SPLINE
SPL {X  -162.820, Y  +621.304, Z    +0.000, E1   +22.259, E3 +582034.378}
SPL {X  -162.820, Y  +618.758, Z    +0.000, E1   +22.239, E3 +582047.529}
SPL {X  -162.820, Y  +616.062, Z    +0.000, E1   +22.275, E3 +582060.950}
SPL {X  -162.820, Y  +613.536, Z    +0.000, E1   +22.242, E3 +582074.071}
SPL {X  -162.820, Y  +610.461, Z    +0.000, E1   +22.264, E3 +582089.703}
SPL {X  -162.820, Y  +606.755, Z    +0.000, E1   +22.275, E3 +582108.501}
SPL {X  -162.820, Y  +603.020, Z    +0.000, E1   +22.272, E3 +582127.561}
SPL {X  -162.820, Y  +599.168, Z    +0.000, E1   +22.310, E3 +582146.829}
SPL {X  -162.820, Y  +595.597, Z    +0.000, E1   +22.284, E3 +582165.165}
SPL {X  -162.820, Y  +593.320, Z    +0.000, E1   +22.199, E3 +582177.255}
SPL {X  -162.820, Y  +591.031, Z    +0.000, E1   +22.283, E3 +582188.346}
SPL {X  -162.820, Y  +588.026, Z    +0.000, E1   +22.301, E3 +582203.473}
SPL {X  -162.820, Y  +585.899, Z    +0.000, E1   +22.286, E3 +582214.275}
SPL {X  -162.820, Y  +583.204, Z    +0.000, E1   +22.278, E3 +582228.298}
SPL {X  -162.820, Y  +579.691, Z    +0.000, E1   +22.312, E3 +582245.786}
SPL {X  -162.820, Y  +576.856, Z    +0.000, E1   +22.233, E3 +582260.836}
SPL {X  -162.820, Y  +574.811, Z    +0.000, E1   +22.236, E3 +582271.100}
SPL {X  -162.820, Y  +572.645, Z    +0.000, E1   +22.246, E3 +582282.195}
SPL {X  -162.820, Y  +569.475, Z    +0.000, E1   +22.269, E3 +582298.202}
SPL {X  -162.820, Y  +565.838, Z    +0.000, E1   +22.271, E3 +582316.796}
SPL {X  -162.820, Y  +562.162, Z    +0.000, E1   +22.252, E3 +582335.614}
SPL {X  -162.820, Y  +558.919, Z    +0.000, E1   +22.286, E3 +582351.777}
SPL {X  -162.820, Y  +556.169, Z    +0.000, E1   +22.295, E3 +582365.606}
SPL {X  -162.820, Y  +553.294, Z    +0.000, E1   +22.266, E3 +582380.604}
SPL {X  -162.820, Y  +550.136, Z    +0.000, E1   +22.258, E3 +582396.717}
SPL {X  -162.820, Y  +546.694, Z    +0.000, E1   +22.290, E3 +582414.039}
SPL {X  -162.820, Y  +543.558, Z    +0.000, E1   +22.285, E3 +582429.902}
SPL {X  -162.820, Y  +541.633, Z    +0.000, E1   +22.257, E3 +582439.830}
SPL {X  -162.820, Y  +539.116, Z    +0.000, E1   +22.302, E3 +582452.441}
SPL {X  -162.820, Y  +535.523, Z    +0.000, E1   +22.266, E3 +582471.103}
SPL {X  -162.820, Y  +531.757, Z    +0.000, E1   +22.276, E3 +582490.157}
SPL {X  -162.820, Y  +527.980, Z    +0.000, E1   +22.326, E3 +582508.988}
SPL {X  -162.820, Y  +524.599, Z    +0.000, E1   +22.287, E3 +582526.385}
SPL {X  -162.820, Y  +522.011, Z    +0.000, E1   +22.282, E3 +582539.462}
SPL {X  -162.820, Y  +519.457, Z    +0.000, E1   +22.481, E3 +582550.752}
SPL {X  -162.820, Y  +505.859, Z    +0.000, E1   +28.367, E3 +582565.235}
SPL {X  -162.820, Y  +504.131, Z    +0.000, E1   +27.325, E3 +582579.373}
SPL {X  -162.820, Y  +503.215, Z    +0.000, E1   +26.369, E3 +582590.059}
SPL {X  -162.820, Y  +502.502, Z    +0.000, E1   +25.597, E3 +582598.906}
SPL {X  -162.820, Y  +501.672, Z    +0.000, E1   +24.583, E3 +582610.521}
SPL {X  -162.820, Y  +500.515, Z    +0.000, E1   +23.444, E3 +582625.051}
SPL {X  -162.820, Y  +499.633, Z    +0.000, E1   +22.486, E3 +582637.097}
SPL {X  -162.820, Y  +498.303, Z    +0.000, E1   +21.749, E3 +582650.406}
SPL {X  -162.820, Y  +495.897, Z    +0.000, E1   +21.662, E3 +582663.560}
SPL {X  -162.820, Y  +493.717, Z    +0.000, E1   +21.704, E3 +582674.666}
SPL {X  -162.820, Y  +491.396, Z    +0.000, E1   +21.707, E3 +582686.790}
SPL {X  -162.820, Y  +489.485, Z    +0.000, E1   +21.661, E3 +582697.138}
SPL {X  -162.820, Y  +487.723, Z    +0.000, E1   +21.665, E3 +582706.342}
SPL {X  -162.820, Y  +485.661, Z    +0.000, E1   +21.712, E3 +582716.785}
SPL {X  -162.820, Y  +482.775, Z    +0.000, E1   +21.716, E3 +582732.037}
SPL {X  -162.820, Y  +479.894, Z    +0.000, E1   +21.695, E3 +582747.114}
SPL {X  -162.820, Y  +477.685, Z    +0.000, E1   +21.656, E3 +582759.051}
SPL {X  -162.820, Y  +475.419, Z    +0.000, E1   +21.711, E3 +582770.404}
SPL {X  -162.820, Y  +473.301, Z    +0.000, E1   +21.712, E3 +582781.501}
SPL {X  -162.820, Y  +470.965, Z    +0.000, E1   +21.700, E3 +582793.846}
SPL {X  -162.820, Y  +469.036, Z    +0.000, E1   +21.695, E3 +582803.890}
SPL {X  -162.820, Y  +467.138, Z    +0.000, E1   +21.678, E3 +582814.061}
SPL {X  -162.820, Y  +465.011, Z    +0.000, E1   +21.692, E3 +582825.044}
SPL {X  -162.820, Y  +462.669, Z    +0.000, E1   +21.752, E3 +582836.824}
SPL {X  -162.820, Y  +460.725, Z    +0.000, E1   +21.689, E3 +582847.437}
SPL {X  -162.820, Y  +458.666, Z    +0.000, E1   +21.695, E3 +582858.249}
SPL {X  -162.820, Y  +456.431, Z    +0.000, E1   +21.708, E3 +582869.778}
SPL {X  -162.820, Y  +454.628, Z    +0.000, E1   +21.674, E3 +582879.496}
SPL {X  -162.820, Y  +452.690, Z    +0.000, E1   +21.773, E3 +582888.770}
SPL {X  -162.820, Y  +450.610, Z    +0.000, E1   +21.698, E3 +582900.369}
SPL {X  -162.820, Y  +448.170, Z    +0.000, E1   +21.667, E3 +582913.390}
SPL {X  -162.820, Y  +446.246, Z    +0.000, E1   +21.696, E3 +582923.208}
SPL {X  -162.820, Y  +443.784, Z    +0.000, E1   +21.713, E3 +582935.994}
SPL {X  -162.820, Y  +440.567, Z    +0.000, E1   +21.731, E3 +582952.834}
SPL {X  -162.820, Y  +437.628, Z    +0.000, E1   +21.678, E3 +582968.498}
SPL {X  -162.820, Y  +435.262, Z    +0.000, E1   +21.727, E3 +582980.433}
SPL {X  -162.820, Y  +433.510, Z    +0.000, E1   +21.692, E3 +582989.847}
SPL {X  -162.820, Y  +431.492, Z    +0.000, E1   +21.686, E3 +583000.543}
SPL {X  -162.820, Y  +429.074, Z    +0.000, E1   +21.710, E3 +583012.995}
SPL {X  -162.820, Y  +427.020, Z    +0.000, E1   +21.674, E3 +583023.996}
SPL {X  -162.820, Y  +424.525, Z    +0.000, E1   +21.712, E3 +583036.909}
SPL {X  -162.820, Y  +421.144, Z    +0.000, E1   +21.719, E3 +583054.576}
SPL {X  -162.820, Y  +418.116, Z    +0.000, E1   +21.761, E3 +583069.907}
SPL {X  -162.820, Y  +416.127, Z    +0.000, E1   +21.715, E3 +583080.612}
SPL {X  -162.820, Y  +414.361, Z    +0.000, E1   +21.613, E3 +583090.800}
SPL {X  -162.820, Y  +412.134, Z    +0.000, E1   +21.697, E3 +583101.744}
SPL {X  -162.820, Y  +409.248, Z    +0.000, E1   +21.741, E3 +583116.679}
SPL {X  -162.820, Y  +406.238, Z    +0.000, E1   +21.697, E3 +583132.647}
SPL {X  -162.820, Y  +404.001, Z    +0.000, E1   +21.723, E3 +583144.077}
SPL {X  -162.820, Y  +402.223, Z    +0.000, E1   +21.697, E3 +583153.562}
SPL {X  -162.820, Y  +400.348, Z    +0.000, E1   +21.713, E3 +583163.288}
SPL {X  -162.820, Y  +398.298, Z    +0.000, E1   +21.721, E3 +583173.904}
SPL {X  -162.820, Y  +396.371, Z    +0.000, E1   +21.713, E3 +583184.086}
SPL {X  -162.820, Y  +394.508, Z    +0.000, E1   +21.616, E3 +583194.641}
SPL {X  -162.820, Y  +392.435, Z    +0.000, E1   +21.681, E3 +583204.994}
SPL {X  -162.820, Y  +389.390, Z    +0.000, E1   +21.742, E3 +583220.601}
SPL {X  -162.820, Y  +386.818, Z    +0.000, E1   +21.679, E3 +583234.360}
SPL {X  -162.820, Y  +384.697, Z    +0.000, E1   +21.693, E3 +583245.430}
SPL {X  -162.820, Y  +382.288, Z    +0.000, E1   +21.742, E3 +583257.554}
SPL {X  -162.817, Y  +379.520, Z    +0.000, E1   +21.723, E3 +583272.391}
SPL {X  -162.776, Y  +376.710, Z    +0.000, E1   +21.698, E3 +583287.130}
SPL {X  -162.707, Y  +374.438, Z    +0.000, E1   +21.688, E3 +583299.134}
SPL {X  -162.607, Y  +372.171, Z    +0.000, E1   +21.692, E3 +583310.934}
SPL {X  -162.494, Y  +370.197, Z    +0.000, E1   +21.655, E3 +583321.560}
SPL {X  -162.349, Y  +368.131, Z    +0.000, E1   +21.624, E3 +583332.678}
SPL {X  -162.161, Y  +365.866, Z    +0.000, E1   +21.642, E3 +583344.363}
SPL {X  -161.651, Y  +361.024, Z    +0.000, E1   +22.970, E3 +583357.787}
SPL {X  -160.281, Y  +351.857, Z    +0.000, E1   +24.243, E3 +583393.126}
ENDSPLINE

SPLINE
SPL {X  -161.833, Y  +362.603, Z    +0.000, E1   +17.021, E3 +583407.822}
ENDSPLINE

SPLINE
SPL {X  -160.786, Y  +354.842, Z    +0.000, E1   +19.274, E3 +583439.977}
ENDSPLINE

SPLINE
SPL {X  -162.485, Y  +370.062, Z    +0.000, E1   +10.606, E3 +583446.355}
SPL {X  -162.818, Y  +379.636, Z    +0.000, E1    +5.115, E3 +583435.704}
SPL {X  -162.820, Y  +386.976, Z    +0.000, E1    +0.144, E3 +583434.803}
SPL {X  -162.820, Y  +391.982, Z    +0.000, E1    -3.443, E3 +583441.568}
SPL {X  -162.820, Y  +399.630, Z    +0.000, E1    -9.426, E3 +583444.076}
SPL {X  -162.820, Y  +408.127, Z    +0.000, E1   -18.417, E3 +583430.364}
SPL {X  -162.820, Y  +420.083, Z    +0.000, E1   -24.325, E3 +583450.839}
SPL {X  -162.820, Y  +428.527, Z    +0.000, E1   -26.988, E3 +583468.132}
SPL {X  -162.820, Y  +431.336, Z    +0.000, E1   -24.162, E3 +583498.342}
SPL {X  -162.820, Y  +432.048, Z    +0.000, E1   -22.832, E3 +583512.845}
SPL {X  -162.820, Y  +434.888, Z    +0.000, E1   -22.823, E3 +583526.795}
SPL {X  -162.820, Y  +436.834, Z    +0.000, E1   -22.779, E3 +583536.755}
SPL {X  -162.820, Y  +438.868, Z    +0.000, E1   -22.837, E3 +583546.408}
SPL {X  -162.820, Y  +441.351, Z    +0.000, E1   -22.805, E3 +583558.984}
SPL {X  -162.820, Y  +443.809, Z    +0.000, E1   -22.804, E3 +583571.150}
SPL {X  -162.820, Y  +446.105, Z    +0.000, E1   -22.815, E3 +583582.392}
SPL {X  -162.820, Y  +447.974, Z    +0.000, E1   -22.856, E3 +583591.295}
SPL {X  -162.820, Y  +449.911, Z    +0.000, E1   -22.774, E3 +583601.570}
SPL {X  -162.820, Y  +451.861, Z    +0.000, E1   -22.750, E3 +583611.417}
SPL {X  -162.820, Y  +454.167, Z    +0.000, E1   -22.842, E3 +583622.147}
SPL {X  -162.820, Y  +456.529, Z    +0.000, E1   -22.855, E3 +583633.675}
SPL {X  -162.820, Y  +458.725, Z    +0.000, E1   -22.793, E3 +583645.080}
SPL {X  -162.820, Y  +461.700, Z    +0.000, E1   -22.822, E3 +583659.702}
SPL {X  -162.820, Y  +464.633, Z    +0.000, E1   -22.813, E3 +583674.199}
SPL {X  -162.820, Y  +466.699, Z    +0.000, E1   -22.824, E3 +583684.245}
SPL {X  -162.820, Y  +468.655, Z    +0.000, E1   -22.858, E3 +583693.689}
SPL {X  -162.820, Y  +470.892, Z    +0.000, E1   -22.837, E3 +583704.927}
SPL {X  -162.820, Y  +473.485, Z    +0.000, E1   -22.806, E3 +583718.126}
SPL {X  -162.820, Y  +476.589, Z    +0.000, E1   -22.788, E3 +583733.648}
SPL {X  -162.820, Y  +478.914, Z    +0.000, E1   -22.821, E3 +583744.746}
SPL {X  -162.820, Y  +481.034, Z    +0.000, E1   -22.831, E3 +583755.268}
SPL {X  -162.820, Y  +484.256, Z    +0.000, E1   -22.840, E3 +583771.287}
SPL {X  -162.820, Y  +487.014, Z    +0.000, E1   -22.789, E3 +583785.154}
SPL {X  -162.820, Y  +489.750, Z    +0.000, E1   -22.832, E3 +583798.528}
SPL {X  -162.820, Y  +493.233, Z    +0.000, E1   -22.844, E3 +583815.665}
SPL {X  -162.820, Y  +496.150, Z    +0.000, E1   -22.796, E3 +583830.384}
SPL {X  -162.820, Y  +498.661, Z    +0.000, E1   -22.828, E3 +583842.565}
SPL {X  -162.820, Y  +501.761, Z    +0.000, E1   -22.820, E3 +583858.134}
SPL {X  -162.820, Y  +505.323, Z    +0.000, E1   -22.838, E3 +583875.581}
SPL {X  -162.820, Y  +507.875, Z    +0.000, E1   -22.849, E3 +583887.948}
SPL {X  -162.820, Y  +510.068, Z    +0.000, E1   -22.761, E3 +583899.641}
SPL {X  -162.820, Y  +512.359, Z    +0.000, E1   -22.823, E3 +583910.372}
SPL {X  -162.820, Y  +514.562, Z    +0.000, E1   -22.806, E3 +583921.559}
SPL {X  -162.820, Y  +517.952, Z    +0.000, E1   -22.864, E3 +583937.957}
SPL {X  -162.820, Y  +520.641, Z    +0.000, E1   -22.790, E3 +583951.675}
SPL {X  -162.820, Y  +522.740, Z    +0.000, E1   -22.811, E3 +583961.918}
SPL {X  -162.820, Y  +524.628, Z    +0.000, E1   -22.846, E3 +583970.913}
SPL {X  -162.820, Y  +526.661, Z    +0.000, E1   -22.801, E3 +583981.468}
SPL {X  -162.820, Y  +529.662, Z    +0.000, E1   -22.810, E3 +583996.319}
SPL {X  -162.820, Y  +532.614, Z    +0.000, E1   -22.828, E3 +584010.725}
SPL {X  -162.820, Y  +534.838, Z    +0.000, E1   -22.864, E3 +584021.354}
SPL {X  -162.820, Y  +536.882, Z    +0.000, E1   -22.782, E3 +584032.209}
SPL {X  -162.820, Y  +539.194, Z    +0.000, E1   -22.826, E3 +584043.257}
SPL {X  -162.820, Y  +541.555, Z    +0.000, E1   -22.817, E3 +584055.072}
SPL {X  -162.820, Y  +543.728, Z    +0.000, E1   -22.799, E3 +584065.929}
SPL {X  -162.820, Y  +545.925, Z    +0.000, E1   -22.803, E3 +584076.799}
SPL {X  -162.820, Y  +549.071, Z    +0.000, E1   -22.836, E3 +584092.326}
SPL {X  -162.820, Y  +553.089, Z    +0.000, E1   -22.838, E3 +584112.226}
SPL {X  -162.820, Y  +556.430, Z    +0.000, E1   -22.821, E3 +584128.728}
SPL {X  -162.820, Y  +558.974, Z    +0.000, E1   -22.806, E3 +584141.428}
SPL {X  -162.820, Y  +562.171, Z    +0.000, E1   -22.845, E3 +584157.126}
SPL {X  -162.820, Y  +565.170, Z    +0.000, E1   -22.801, E3 +584172.139}
SPL {X  -162.820, Y  +567.308, Z    +0.000, E1   -22.750, E3 +584183.155}
SPL {X  -162.820, Y  +570.378, Z    +0.000, E1   -22.843, E3 +584197.779}
SPL {X  -162.820, Y  +573.634, Z    +0.000, E1   -22.827, E3 +584213.923}
SPL {X  -162.820, Y  +576.228, Z    +0.000, E1   -22.814, E3 +584226.819}
SPL {X  -162.820, Y  +578.553, Z    +0.000, E1   -22.801, E3 +584238.435}
SPL {X  -162.820, Y  +581.064, Z    +0.000, E1   -22.823, E3 +584250.719}
SPL {X  -162.820, Y  +583.435, Z    +0.000, E1   -22.808, E3 +584262.541}
SPL {X  -162.820, Y  +585.410, Z    +0.000, E1   -22.764, E3 +584272.677}
SPL {X  -162.820, Y  +587.676, Z    +0.000, E1   -22.853, E3 +584283.191}
SPL {X  -162.820, Y  +590.707, Z    +0.000, E1   -22.855, E3 +584298.342}
SPL {X  -162.820, Y  +593.650, Z    +0.000, E1   -22.810, E3 +584313.102}
SPL {X  -162.820, Y  +595.830, Z    +0.000, E1   -22.828, E3 +584323.718}
SPL {X  -162.820, Y  +598.094, Z    +0.000, E1   -22.843, E3 +584334.831}
SPL {X  -162.820, Y  +600.420, Z    +0.000, E1   -22.826, E3 +584346.462}
SPL {X  -162.820, Y  +602.573, Z    +0.000, E1   -22.830, E3 +584357.047}
SPL {X  -162.820, Y  +604.828, Z    +0.000, E1   -22.784, E3 +584368.686}
SPL {X  -162.820, Y  +608.133, Z    +0.000, E1   -22.831, E3 +584384.803}
SPL {X  -162.820, Y  +611.103, Z    +0.000, E1   -22.785, E3 +584399.729}
SPL {X  -162.820, Y  +613.294, Z    +0.000, E1   -22.780, E3 +584410.602}
SPL {X  -162.820, Y  +615.356, Z    +0.000, E1   -22.799, E3 +584420.660}
SPL {X  -162.820, Y  +617.439, Z    +0.000, E1   -22.808, E3 +584430.918}
SPL {X  -162.820, Y  +619.665, Z    +0.000, E1   -22.817, E3 +584441.886}
SPL {X  -162.820, Y  +621.733, Z    +0.000, E1   -22.759, E3 +584452.610}
SPL {X  -162.820, Y  +624.076, Z    +0.000, E1   -22.774, E3 +584464.115}
SPL {X  -162.820, Y  +626.527, Z    +0.000, E1   -22.768, E3 +584476.358}
SPL {X  -162.820, Y  +629.758, Z    +0.000, E1   -22.800, E3 +584492.286}
SPL {X  -162.820, Y  +632.572, Z    +0.000, E1   -22.785, E3 +584506.136}
SPL {X  -162.820, Y  +634.507, Z    +0.000, E1   -22.784, E3 +584515.775}
SPL {X  -162.820, Y  +636.863, Z    +0.000, E1   -22.760, E3 +584527.697}
SPL {X  -162.820, Y  +639.254, Z    +0.000, E1   -22.767, E3 +584539.480}
SPL {X  -162.820, Y  +641.888, Z    +0.000, E1   -22.790, E3 +584552.427}
SPL {X  -162.820, Y  +644.915, Z    +0.000, E1   -22.818, E3 +584567.202}
SPL {X  -162.820, Y  +647.561, Z    +0.000, E1   -22.705, E3 +584581.244}
SPL {X  -162.820, Y  +649.758, Z    +0.000, E1   -22.780, E3 +584591.434}
SPL {X  -162.820, Y  +651.708, Z    +0.000, E1   -22.810, E3 +584600.929}
SPL {X  -162.820, Y  +653.898, Z    +0.000, E1   -22.796, E3 +584611.849}
SPL {X  -162.820, Y  +656.161, Z    +0.000, E1   -22.812, E3 +584622.971}
SPL {X  -162.820, Y  +658.384, Z    +0.000, E1   -22.822, E3 +584633.837}
SPL {X  -162.820, Y  +660.215, Z    +0.000, E1   -22.649, E3 +584644.428}
SPL {X  -162.820, Y  +662.823, Z    +0.000, E1   -22.799, E3 +584656.136}
SPL {X  -162.820, Y  +665.862, Z    +0.000, E1   -22.864, E3 +584670.835}
SPL {X  -162.820, Y  +668.960, Z    +0.000, E1   -22.773, E3 +584686.786}
SPL {X  -162.820, Y  +671.605, Z    +0.000, E1   -22.777, E3 +584699.860}
SPL {X  -162.817, Y  +674.515, Z    +0.000, E1   -22.816, E3 +584714.057}
SPL {X  -162.773, Y  +677.428, Z    +0.000, E1   -22.762, E3 +584728.865}
SPL {X  -162.691, Y  +679.987, Z    +0.000, E1   -22.794, E3 +584741.278}
SPL {X  -162.559, Y  +682.717, Z    +0.000, E1   -22.726, E3 +584755.461}
SPL {X  -162.404, Y  +685.137, Z    +0.000, E1   -22.766, E3 +584766.984}
SPL {X  -162.229, Y  +687.364, Z    +0.000, E1   -22.685, E3 +584778.852}
SPL {X  -161.938, Y  +690.422, Z    +0.000, E1   -22.769, E3 +584793.258}
SPL {X  -161.065, Y  +697.344, Z    +0.000, E1   -25.698, E3 +584802.378}
SPL {X  -158.553, Y  +710.529, Z    +0.000, E1   -30.890, E3 +584816.274}
ENDSPLINE

SPLINE
SPL {X  -161.215, Y  +696.305, Z    +0.000, E1   -20.575, E3 +584842.855}
SPL {X  -161.691, Y  +692.643, Z    +0.000, E1   -17.369, E3 +584859.043}
SPL {X  -162.534, Y  +683.153, Z    +0.000, E1   -10.475, E3 +584884.510}
SPL {X  -162.820, Y  +670.105, Z    +0.000, E1    -2.484, E3 +584877.157}
SPL {X  -162.820, Y  +665.819, Z    +0.000, E1    +0.492, E3 +584879.453}
SPL {X  -162.820, Y  +661.883, Z    +0.000, E1    +3.373, E3 +584883.930}
SPL {X  -162.820, Y  +655.163, Z    +0.000, E1    +8.702, E3 +584883.529}
SPL {X  -162.820, Y  +634.515, Z    +0.000, E1   +26.439, E3 +584875.942}
ENDSPLINE

SPLINE
SPL {X  -162.820, Y  +638.080, Z    +0.000, E1   +18.858, E3 +584905.906}
ENDSPLINE

SPLINE
SPL {X  -162.820, Y  +623.278, Z    +0.000, E1   +28.723, E3 +584907.477}
SPL {X  -162.820, Y  +611.829, Z    +0.000, E1   +31.229, E3 +584931.129}
ENDSPLINE

SPLINE
SPL {X  -162.820, Y  +623.595, Z    +0.000, E1   +22.712, E3 +584946.050}
ENDSPLINE

SPLINE
SPL {X  -162.820, Y  +621.304, Z    +0.000, E1   +22.259, E3 +584961.208}
SPL {X  -162.820, Y  +618.758, Z    +0.000, E1   +22.239, E3 +584974.358}
SPL {X  -162.820, Y  +616.062, Z    +0.000, E1   +22.275, E3 +584987.779}
SPL {X  -162.820, Y  +613.536, Z    +0.000, E1   +22.242, E3 +585000.901}
SPL {X  -162.820, Y  +611.128, Z    +0.000, E1   +22.252, E3 +585013.071}
SPL {X  -162.820, Y  +608.428, Z    +0.000, E1   +22.255, E3 +585026.855}
SPL {X  -162.820, Y  +605.178, Z    +0.000, E1   +22.267, E3 +585043.387}
SPL {X  -162.820, Y  +602.350, Z    +0.000, E1   +22.224, E3 +585058.004}
SPL {X  -162.820, Y  +599.842, Z    +0.000, E1   +22.298, E3 +585070.156}
SPL {X  -162.820, Y  +597.194, Z    +0.000, E1   +22.253, E3 +585084.077}
SPL {X  -162.820, Y  +594.779, Z    +0.000, E1   +22.284, E3 +585095.980}
SPL {X  -162.820, Y  +592.389, Z    +0.000, E1   +22.245, E3 +585108.597}
SPL {X  -162.820, Y  +589.492, Z    +0.000, E1   +22.304, E3 +585122.781}
SPL {X  -162.820, Y  +587.447, Z    +0.000, E1   +22.279, E3 +585133.310}
SPL {X  -162.820, Y  +585.192, Z    +0.000, E1   +22.298, E3 +585144.721}
SPL {X  -162.820, Y  +582.610, Z    +0.000, E1   +22.234, E3 +585158.344}
SPL {X  -162.820, Y  +580.317, Z    +0.000, E1   +22.300, E3 +585169.398}
SPL {X  -162.820, Y  +578.878, Z    +0.000, E1   +22.272, E3 +585176.907}
SPL {X  -162.820, Y  +576.856, Z    +0.000, E1   +22.233, E3 +585187.666}
SPL {X  -162.820, Y  +574.811, Z    +0.000, E1   +22.236, E3 +585197.929}
SPL {X  -162.820, Y  +572.645, Z    +0.000, E1   +22.246, E3 +585209.025}
SPL {X  -162.820, Y  +569.475, Z    +0.000, E1   +22.269, E3 +585225.031}
SPL {X  -162.820, Y  +565.838, Z    +0.000, E1   +22.271, E3 +585243.626}
SPL {X  -162.820, Y  +562.162, Z    +0.000, E1   +22.252, E3 +585262.443}
SPL {X  -162.820, Y  +558.919, Z    +0.000, E1   +22.286, E3 +585278.606}
SPL {X  -162.820, Y  +556.169, Z    +0.000, E1   +22.295, E3 +585292.436}
SPL {X  -162.820, Y  +553.294, Z    +0.000, E1   +22.266, E3 +585307.433}
SPL {X  -162.820, Y  +550.136, Z    +0.000, E1   +22.258, E3 +585323.546}
SPL {X  -162.820, Y  +546.694, Z    +0.000, E1   +22.290, E3 +585340.868}
SPL {X  -162.820, Y  +543.558, Z    +0.000, E1   +22.285, E3 +585356.731}
SPL {X  -162.820, Y  +541.633, Z    +0.000, E1   +22.257, E3 +585366.659}
SPL {X  -162.820, Y  +539.116, Z    +0.000, E1   +22.302, E3 +585379.270}
SPL {X  -162.820, Y  +536.913, Z    +0.000, E1   +22.192, E3 +585391.195}
SPL {X  -162.820, Y  +534.880, Z    +0.000, E1   +22.252, E3 +585401.148}
SPL {X  -162.820, Y  +532.896, Z    +0.000, E1   +22.234, E3 +585411.308}
SPL {X  -162.820, Y  +531.056, Z    +0.000, E1   +22.251, E3 +585420.590}
SPL {X  -162.820, Y  +528.708, Z    +0.000, E1   +22.319, E3 +585431.972}
SPL {X  -162.820, Y  +525.932, Z    +0.000, E1   +22.258, E3 +585446.728}
SPL {X  -162.820, Y  +522.524, Z    +0.000, E1   +22.326, E3 +585463.452}
SPL {X  -162.820, Y  +519.457, Z    +0.000, E1   +22.481, E3 +585477.581}
SPL {X  -162.820, Y  +506.285, Z    +0.000, E1   +28.538, E3 +585489.039}
SPL {X  -162.820, Y  +504.441, Z    +0.000, E1   +27.574, E3 +585503.381}
SPL {X  -162.820, Y  +502.813, Z    +0.000, E1   +26.013, E3 +585521.579}
SPL {X  -162.820, Y  +502.016, Z    +0.000, E1   +24.802, E3 +585533.921}
SPL {X  -162.820, Y  +501.060, Z    +0.000, E1   +24.081, E3 +585544.111}
SPL {X  -162.820, Y  +500.336, Z    +0.000, E1   +23.110, E3 +585555.251}
SPL {X  -162.820, Y  +499.240, Z    +0.000, E1   +22.316, E3 +585567.561}
SPL {X  -162.820, Y  +498.027, Z    +0.000, E1   +21.516, E3 +585580.469}
SPL {X  -162.820, Y  +495.897, Z    +0.000, E1   +21.662, E3 +585590.389}
SPL {X  -162.820, Y  +493.717, Z    +0.000, E1   +21.704, E3 +585601.496}
SPL {X  -162.820, Y  +491.396, Z    +0.000, E1   +21.707, E3 +585613.620}
SPL {X  -162.820, Y  +488.560, Z    +0.000, E1   +21.695, E3 +585628.729}
SPL {X  -162.820, Y  +485.661, Z    +0.000, E1   +21.712, E3 +585643.614}
SPL {X  -162.820, Y  +483.668, Z    +0.000, E1   +21.664, E3 +585654.442}
SPL {X  -162.820, Y  +481.739, Z    +0.000, E1   +21.704, E3 +585664.156}
SPL {X  -162.820, Y  +479.894, Z    +0.000, E1   +21.695, E3 +585673.943}
SPL {X  -162.820, Y  +477.685, Z    +0.000, E1   +21.656, E3 +585685.881}
SPL {X  -162.820, Y  +475.419, Z    +0.000, E1   +21.711, E3 +585697.233}
SPL {X  -162.820, Y  +473.301, Z    +0.000, E1   +21.712, E3 +585708.330}
SPL {X  -162.820, Y  +470.965, Z    +0.000, E1   +21.700, E3 +585720.675}
SPL {X  -162.820, Y  +469.036, Z    +0.000, E1   +21.695, E3 +585730.719}
SPL {X  -162.820, Y  +467.138, Z    +0.000, E1   +21.678, E3 +585740.891}
SPL {X  -162.820, Y  +465.011, Z    +0.000, E1   +21.692, E3 +585751.873}
SPL {X  -162.820, Y  +462.669, Z    +0.000, E1   +21.752, E3 +585763.654}
SPL {X  -162.820, Y  +460.725, Z    +0.000, E1   +21.689, E3 +585774.267}
SPL {X  -162.820, Y  +458.666, Z    +0.000, E1   +21.695, E3 +585785.079}
SPL {X  -162.820, Y  +456.431, Z    +0.000, E1   +21.708, E3 +585796.607}
SPL {X  -162.820, Y  +453.609, Z    +0.000, E1   +21.757, E3 +585811.141}
SPL {X  -162.820, Y  +450.610, Z    +0.000, E1   +21.698, E3 +585827.198}
SPL {X  -162.820, Y  +448.170, Z    +0.000, E1   +21.667, E3 +585840.219}
SPL {X  -162.820, Y  +446.246, Z    +0.000, E1   +21.696, E3 +585850.037}
SPL {X  -162.820, Y  +443.784, Z    +0.000, E1   +21.713, E3 +585862.823}
SPL {X  -162.820, Y  +440.567, Z    +0.000, E1   +21.731, E3 +585879.663}
SPL {X  -162.820, Y  +437.628, Z    +0.000, E1   +21.678, E3 +585895.327}
SPL {X  -162.820, Y  +434.473, Z    +0.000, E1   +21.747, E3 +585911.423}
SPL {X  -162.820, Y  +431.492, Z    +0.000, E1   +21.686, E3 +585927.372}
SPL {X  -162.820, Y  +429.074, Z    +0.000, E1   +21.710, E3 +585939.824}
SPL {X  -162.820, Y  +426.023, Z    +0.000, E1   +21.718, E3 +585955.892}
SPL {X  -162.820, Y  +422.986, Z    +0.000, E1   +21.685, E3 +585971.939}
SPL {X  -162.820, Y  +420.528, Z    +0.000, E1   +21.706, E3 +585984.589}
SPL {X  -162.820, Y  +418.116, Z    +0.000, E1   +21.761, E3 +585996.736}
SPL {X  -162.820, Y  +416.127, Z    +0.000, E1   +21.715, E3 +586007.442}
SPL {X  -162.820, Y  +414.361, Z    +0.000, E1   +21.613, E3 +586017.629}
SPL {X  -162.820, Y  +411.450, Z    +0.000, E1   +21.710, E3 +586032.202}
SPL {X  -162.820, Y  +408.590, Z    +0.000, E1   +21.735, E3 +586046.828}
SPL {X  -162.820, Y  +406.238, Z    +0.000, E1   +21.697, E3 +586059.477}
SPL {X  -162.820, Y  +403.166, Z    +0.000, E1   +21.746, E3 +586075.283}
SPL {X  -162.820, Y  +400.348, Z    +0.000, E1   +21.713, E3 +586090.117}
SPL {X  -162.820, Y  +398.298, Z    +0.000, E1   +21.721, E3 +586100.733}
SPL {X  -162.820, Y  +396.371, Z    +0.000, E1   +21.713, E3 +586110.915}
SPL {X  -162.820, Y  +394.508, Z    +0.000, E1   +21.616, E3 +586121.470}
SPL {X  -162.820, Y  +391.777, Z    +0.000, E1   +21.714, E3 +586135.130}
SPL {X  -162.820, Y  +388.822, Z    +0.000, E1   +21.717, E3 +586150.449}
SPL {X  -162.820, Y  +386.818, Z    +0.000, E1   +21.679, E3 +586161.189}
SPL {X  -162.820, Y  +384.697, Z    +0.000, E1   +21.693, E3 +586172.260}
SPL {X  -162.820, Y  +382.288, Z    +0.000, E1   +21.742, E3 +586184.383}
SPL {X  -162.820, Y  +380.381, Z    +0.000, E1   +21.655, E3 +586195.108}
SPL {X  -162.808, Y  +378.512, Z    +0.000, E1   +21.736, E3 +586204.160}
SPL {X  -162.776, Y  +376.710, Z    +0.000, E1   +21.698, E3 +586213.960}
SPL {X  -162.707, Y  +374.438, Z    +0.000, E1   +21.688, E3 +586225.964}
SPL {X  -162.607, Y  +372.171, Z    +0.000, E1   +21.692, E3 +586237.763}
SPL {X  -162.494, Y  +370.197, Z    +0.000, E1   +21.655, E3 +586248.389}
SPL {X  -162.349, Y  +368.131, Z    +0.000, E1   +21.624, E3 +586259.507}
SPL {X  -162.161, Y  +365.866, Z    +0.000, E1   +21.642, E3 +586271.193}
SPL {X  -161.651, Y  +361.024, Z    +0.000, E1   +22.970, E3 +586284.616}
SPL {X  -160.281, Y  +351.857, Z    +0.000, E1   +24.243, E3 +586319.955}
ENDSPLINE

SPLINE
SPL {X  -161.833, Y  +362.603, Z    +0.000, E1   +17.021, E3 +586334.651}
ENDSPLINE

SPLINE
SPL {X  -160.786, Y  +354.842, Z    +0.000, E1   +19.274, E3 +586366.806}
ENDSPLINE

SPLINE
SPL {X  -162.485, Y  +370.062, Z    +0.000, E1   +10.606, E3 +586373.185}
SPL {X  -162.818, Y  +379.636, Z    +0.000, E1    +5.115, E3 +586362.534}
SPL {X  -162.820, Y  +386.976, Z    +0.000, E1    +0.144, E3 +586361.633}
SPL {X  -162.820, Y  +391.982, Z    +0.000, E1    -3.443, E3 +586368.397}
SPL {X  -162.820, Y  +399.630, Z    +0.000, E1    -9.426, E3 +586370.905}
SPL {X  -162.820, Y  +408.127, Z    +0.000, E1   -18.417, E3 +586357.193}
SPL {X  -162.820, Y  +420.083, Z    +0.000, E1   -24.325, E3 +586377.669}
SPL {X  -162.820, Y  +428.527, Z    +0.000, E1   -26.988, E3 +586394.961}
SPL {X  -162.820, Y  +431.191, Z    +0.000, E1   -23.548, E3 +586429.814}
SPL {X  -162.820, Y  +432.946, Z    +0.000, E1   -22.795, E3 +586444.217}
SPL {X  -162.820, Y  +434.888, Z    +0.000, E1   -22.823, E3 +586453.624}
SPL {X  -162.820, Y  +436.834, Z    +0.000, E1   -22.779, E3 +586463.584}
SPL {X  -162.820, Y  +438.868, Z    +0.000, E1   -22.837, E3 +586473.238}
SPL {X  -162.820, Y  +441.351, Z    +0.000, E1   -22.805, E3 +586485.813}
SPL {X  -162.820, Y  +443.809, Z    +0.000, E1   -22.804, E3 +586497.979}
SPL {X  -162.820, Y  +447.077, Z    +0.000, E1   -22.869, E3 +586513.790}
SPL {X  -162.820, Y  +449.911, Z    +0.000, E1   -22.774, E3 +586528.399}
SPL {X  -162.820, Y  +451.861, Z    +0.000, E1   -22.750, E3 +586538.247}
SPL {X  -162.820, Y  +454.167, Z    +0.000, E1   -22.842, E3 +586548.976}
SPL {X  -162.820, Y  +456.529, Z    +0.000, E1   -22.855, E3 +586560.505}
SPL {X  -162.820, Y  +458.725, Z    +0.000, E1   -22.793, E3 +586571.909}
SPL {X  -162.820, Y  +461.700, Z    +0.000, E1   -22.822, E3 +586586.532}
SPL {X  -162.820, Y  +464.633, Z    +0.000, E1   -22.813, E3 +586601.028}
SPL {X  -162.820, Y  +466.699, Z    +0.000, E1   -22.824, E3 +586611.074}
SPL {X  -162.820, Y  +468.655, Z    +0.000, E1   -22.858, E3 +586620.518}
SPL {X  -162.820, Y  +470.892, Z    +0.000, E1   -22.837, E3 +586631.757}
SPL {X  -162.820, Y  +473.485, Z    +0.000, E1   -22.806, E3 +586644.955}
SPL {X  -162.820, Y  +475.738, Z    +0.000, E1   -22.728, E3 +586656.620}
SPL {X  -162.820, Y  +478.177, Z    +0.000, E1   -22.834, E3 +586667.960}
SPL {X  -162.820, Y  +481.034, Z    +0.000, E1   -22.831, E3 +586682.097}
SPL {X  -162.820, Y  +483.391, Z    +0.000, E1   -22.793, E3 +586694.033}
SPL {X  -162.820, Y  +486.307, Z    +0.000, E1   -22.833, E3 +586708.287}
SPL {X  -162.820, Y  +489.750, Z    +0.000, E1   -22.832, E3 +586725.357}
SPL {X  -162.820, Y  +492.546, Z    +0.000, E1   -22.823, E3 +586739.115}
SPL {X  -162.820, Y  +495.526, Z    +0.000, E1   -22.833, E3 +586753.998}
SPL {X  -162.820, Y  +499.330, Z    +0.000, E1   -22.841, E3 +586772.779}
SPL {X  -162.820, Y  +503.049, Z    +0.000, E1   -22.823, E3 +586791.329}
SPL {X  -162.820, Y  +506.908, Z    +0.000, E1   -22.877, E3 +586809.999}
SPL {X  -162.820, Y  +510.068, Z    +0.000, E1   -22.761, E3 +586826.470}
SPL {X  -162.820, Y  +512.359, Z    +0.000, E1   -22.823, E3 +586837.202}
SPL {X  -162.820, Y  +513.873, Z    +0.000, E1   -22.800, E3 +586844.888}
SPL {X  -162.820, Y  +516.100, Z    +0.000, E1   -22.809, E3 +586855.965}
SPL {X  -162.820, Y  +518.662, Z    +0.000, E1   -22.847, E3 +586868.263}
SPL {X  -162.820, Y  +520.641, Z    +0.000, E1   -22.790, E3 +586878.504}
SPL {X  -162.820, Y  +523.535, Z    +0.000, E1   -22.857, E3 +586892.473}
SPL {X  -162.820, Y  +526.661, Z    +0.000, E1   -22.801, E3 +586908.297}
SPL {X  -162.820, Y  +528.725, Z    +0.000, E1   -22.770, E3 +586918.667}
SPL {X  -162.820, Y  +530.303, Z    +0.000, E1   -22.798, E3 +586926.286}
SPL {X  -162.820, Y  +532.614, Z    +0.000, E1   -22.828, E3 +586937.554}
SPL {X  -162.820, Y  +534.838, Z    +0.000, E1   -22.864, E3 +586948.183}
SPL {X  -162.820, Y  +536.882, Z    +0.000, E1   -22.782, E3 +586959.038}
SPL {X  -162.820, Y  +539.194, Z    +0.000, E1   -22.826, E3 +586970.087}
SPL {X  -162.820, Y  +541.555, Z    +0.000, E1   -22.817, E3 +586981.901}
SPL {X  -162.820, Y  +543.728, Z    +0.000, E1   -22.799, E3 +586992.758}
SPL {X  -162.820, Y  +545.925, Z    +0.000, E1   -22.803, E3 +587003.628}
SPL {X  -162.820, Y  +548.328, Z    +0.000, E1   -22.796, E3 +587015.624}
SPL {X  -162.820, Y  +551.027, Z    +0.000, E1   -22.819, E3 +587028.817}
SPL {X  -162.820, Y  +553.721, Z    +0.000, E1   -22.807, E3 +587042.261}
SPL {X  -162.820, Y  +556.430, Z    +0.000, E1   -22.821, E3 +587055.557}
SPL {X  -162.820, Y  +559.675, Z    +0.000, E1   -22.837, E3 +587071.637}
SPL {X  -162.820, Y  +562.799, Z    +0.000, E1   -22.814, E3 +587087.143}
SPL {X  -162.820, Y  +565.170, Z    +0.000, E1   -22.801, E3 +587098.968}
SPL {X  -162.820, Y  +568.020, Z    +0.000, E1   -22.787, E3 +587113.355}
SPL {X  -162.820, Y  +570.992, Z    +0.000, E1   -22.834, E3 +587127.574}
SPL {X  -162.820, Y  +572.901, Z    +0.000, E1   -22.775, E3 +587137.442}
SPL {X  -162.820, Y  +575.638, Z    +0.000, E1   -22.855, E3 +587150.552}
SPL {X  -162.820, Y  +578.553, Z    +0.000, E1   -22.801, E3 +587165.264}
SPL {X  -162.820, Y  +581.064, Z    +0.000, E1   -22.823, E3 +587177.549}
SPL {X  -162.820, Y  +583.435, Z    +0.000, E1   -22.808, E3 +587189.370}
SPL {X  -162.820, Y  +585.410, Z    +0.000, E1   -22.764, E3 +587199.506}
SPL {X  -162.820, Y  +587.676, Z    +0.000, E1   -22.853, E3 +587210.021}
SPL {X  -162.820, Y  +589.682, Z    +0.000, E1   -22.776, E3 +587220.551}
SPL {X  -162.820, Y  +591.720, Z    +0.000, E1   -22.868, E3 +587229.861}
SPL {X  -162.820, Y  +593.650, Z    +0.000, E1   -22.810, E3 +587239.931}
SPL {X  -162.820, Y  +595.830, Z    +0.000, E1   -22.828, E3 +587250.547}
SPL {X  -162.820, Y  +598.094, Z    +0.000, E1   -22.843, E3 +587261.660}
SPL {X  -162.820, Y  +600.420, Z    +0.000, E1   -22.826, E3 +587273.291}
SPL {X  -162.820, Y  +602.573, Z    +0.000, E1   -22.830, E3 +587283.877}
SPL {X  -162.820, Y  +604.828, Z    +0.000, E1   -22.784, E3 +587295.515}
SPL {X  -162.820, Y  +608.133, Z    +0.000, E1   -22.831, E3 +587311.633}
SPL {X  -162.820, Y  +611.103, Z    +0.000, E1   -22.785, E3 +587326.558}
SPL {X  -162.820, Y  +613.294, Z    +0.000, E1   -22.780, E3 +587337.432}
SPL {X  -162.820, Y  +615.356, Z    +0.000, E1   -22.799, E3 +587347.489}
SPL {X  -162.820, Y  +617.439, Z    +0.000, E1   -22.808, E3 +587357.747}
SPL {X  -162.820, Y  +619.665, Z    +0.000, E1   -22.817, E3 +587368.715}
SPL {X  -162.820, Y  +621.733, Z    +0.000, E1   -22.759, E3 +587379.439}
SPL {X  -162.820, Y  +624.076, Z    +0.000, E1   -22.774, E3 +587390.944}
SPL {X  -162.820, Y  +627.244, Z    +0.000, E1   -22.803, E3 +587406.627}
SPL {X  -162.820, Y  +630.349, Z    +0.000, E1   -22.766, E3 +587422.158}
SPL {X  -162.820, Y  +632.572, Z    +0.000, E1   -22.785, E3 +587432.965}
SPL {X  -162.820, Y  +634.507, Z    +0.000, E1   -22.784, E3 +587442.604}
SPL {X  -162.820, Y  +636.863, Z    +0.000, E1   -22.760, E3 +587454.526}
SPL {X  -162.820, Y  +639.254, Z    +0.000, E1   -22.767, E3 +587466.309}
SPL {X  -162.820, Y  +641.195, Z    +0.000, E1   -22.782, E3 +587475.757}
SPL {X  -162.820, Y  +643.449, Z    +0.000, E1   -22.796, E3 +587486.927}
SPL {X  -162.820, Y  +645.630, Z    +0.000, E1   -22.795, E3 +587497.623}
SPL {X  -162.820, Y  +647.561, Z    +0.000, E1   -22.705, E3 +587508.073}
SPL {X  -162.820, Y  +651.051, Z    +0.000, E1   -22.833, E3 +587524.493}
SPL {X  -162.820, Y  +653.898, Z    +0.000, E1   -22.796, E3 +587538.679}
SPL {X  -162.820, Y  +656.161, Z    +0.000, E1   -22.812, E3 +587549.800}
SPL {X  -162.820, Y  +658.384, Z    +0.000, E1   -22.822, E3 +587560.666}
SPL {X  -162.820, Y  +660.215, Z    +0.000, E1   -22.649, E3 +587571.257}
SPL {X  -162.820, Y  +662.823, Z    +0.000, E1   -22.799, E3 +587582.965}
SPL {X  -162.820, Y  +665.112, Z    +0.000, E1   -22.835, E3 +587594.019}
SPL {X  -162.820, Y  +667.016, Z    +0.000, E1   -22.823, E3 +587603.448}
SPL {X  -162.820, Y  +668.960, Z    +0.000, E1   -22.773, E3 +587613.615}
SPL {X  -162.820, Y  +671.605, Z    +0.000, E1   -22.777, E3 +587626.689}
SPL {X  -162.817, Y  +674.515, Z    +0.000, E1   -22.816, E3 +587640.886}
SPL {X  -162.773, Y  +677.428, Z    +0.000, E1   -22.762, E3 +587655.694}
SPL {X  -162.691, Y  +679.987, Z    +0.000, E1   -22.794, E3 +587668.107}
SPL {X  -162.604, Y  +681.880, Z    +0.000, E1   -22.691, E3 +587678.268}
SPL {X  -162.458, Y  +684.346, Z    +0.000, E1   -22.764, E3 +587690.062}
SPL {X  -162.296, Y  +686.547, Z    +0.000, E1   -22.660, E3 +587701.678}
SPL {X  -162.090, Y  +688.902, Z    +0.000, E1   -22.700, E3 +587713.187}
SPL {X  -161.474, Y  +694.390, Z    +0.000, E1   -24.298, E3 +587726.542}
SPL {X  -158.730, Y  +709.763, Z    +0.000, E1   -31.225, E3 +587737.880}
ENDSPLINE

SPLINE
SPL {X  -160.932, Y  +698.225, Z    +0.000, E1   -21.712, E3 +587768.990}
SPL {X  -161.691, Y  +692.643, Z    +0.000, E1   -17.369, E3 +587785.873}
SPL {X  -162.534, Y  +683.153, Z    +0.000, E1   -10.475, E3 +587811.340}
SPL {X  -162.820, Y  +670.105, Z    +0.000, E1    -2.484, E3 +587803.986}
SPL {X  -162.820, Y  +665.819, Z    +0.000, E1    +0.492, E3 +587806.283}
SPL {X  -162.820, Y  +661.883, Z    +0.000, E1    +3.373, E3 +587810.759}
SPL {X  -162.820, Y  +653.808, Z    +0.000, E1    +9.891, E3 +587808.450}
SPL {X  -162.820, Y  +632.548, Z    +0.000, E1   +27.446, E3 +587804.987}
ENDSPLINE

SPLINE
SPL {X  -162.820, Y  +638.080, Z    +0.000, E1   +18.858, E3 +587832.736}
ENDSPLINE

SPLINE
SPL {X  -162.820, Y  +623.278, Z    +0.000, E1   +28.723, E3 +587834.306}
SPL {X  -162.820, Y  +611.829, Z    +0.000, E1   +31.229, E3 +587857.958}
ENDSPLINE

SPLINE
SPL {X  -162.820, Y  +623.595, Z    +0.000, E1   +22.712, E3 +587872.879}
ENDSPLINE

SPLINE
SPL {X  -162.820, Y  +621.304, Z    +0.000, E1   +22.259, E3 +587888.037}
SPL {X  -162.820, Y  +618.758, Z    +0.000, E1   +22.239, E3 +587901.188}
SPL {X  -162.820, Y  +616.062, Z    +0.000, E1   +22.275, E3 +587914.608}
SPL {X  -162.820, Y  +613.536, Z    +0.000, E1   +22.242, E3 +587927.730}
SPL {X  -162.820, Y  +610.461, Z    +0.000, E1   +22.264, E3 +587943.361}
SPL {X  -162.820, Y  +606.755, Z    +0.000, E1   +22.275, E3 +587962.159}
SPL {X  -162.820, Y  +603.020, Z    +0.000, E1   +22.272, E3 +587981.219}
SPL {X  -162.820, Y  +599.168, Z    +0.000, E1   +22.310, E3 +588000.487}
SPL {X  -162.820, Y  +596.569, Z    +0.000, E1   +22.222, E3 +588014.209}
SPL {X  -162.820, Y  +594.115, Z    +0.000, E1   +22.273, E3 +588026.435}
SPL {X  -162.820, Y  +591.721, Z    +0.000, E1   +22.239, E3 +588038.750}
SPL {X  -162.820, Y  +589.492, Z    +0.000, E1   +22.304, E3 +588049.611}
SPL {X  -162.820, Y  +586.660, Z    +0.000, E1   +22.307, E3 +588064.051}
SPL {X  -162.820, Y  +583.204, Z    +0.000, E1   +22.278, E3 +588081.956}
SPL {X  -162.820, Y  +580.317, Z    +0.000, E1   +22.300, E3 +588096.227}
SPL {X  -162.820, Y  +578.061, Z    +0.000, E1   +22.264, E3 +588108.112}
SPL {X  -162.820, Y  +575.394, Z    +0.000, E1   +22.240, E3 +588121.857}
SPL {X  -162.820, Y  +573.156, Z    +0.000, E1   +22.254, E3 +588133.066}
SPL {X  -162.820, Y  +570.852, Z    +0.000, E1   +22.234, E3 +588145.090}
SPL {X  -162.820, Y  +567.961, Z    +0.000, E1   +22.247, E3 +588159.694}
SPL {X  -162.820, Y  +564.506, Z    +0.000, E1   +22.298, E3 +588177.008}
SPL {X  -162.820, Y  +561.620, Z    +0.000, E1   +22.191, E3 +588192.389}
SPL {X  -162.820, Y  +559.515, Z    +0.000, E1   +22.273, E3 +588202.391}
SPL {X  -162.820, Y  +556.723, Z    +0.000, E1   +22.309, E3 +588216.475}
SPL {X  -162.820, Y  +553.294, Z    +0.000, E1   +22.266, E3 +588234.262}
SPL {X  -162.820, Y  +550.871, Z    +0.000, E1   +22.229, E3 +588246.736}
SPL {X  -162.820, Y  +548.168, Z    +0.000, E1   +22.298, E3 +588260.073}
SPL {X  -162.820, Y  +545.860, Z    +0.000, E1   +22.216, E3 +588272.330}
SPL {X  -162.820, Y  +543.558, Z    +0.000, E1   +22.285, E3 +588283.561}
SPL {X  -162.820, Y  +540.968, Z    +0.000, E1   +22.274, E3 +588296.833}
SPL {X  -162.820, Y  +538.512, Z    +0.000, E1   +22.287, E3 +588309.145}
SPL {X  -162.820, Y  +535.523, Z    +0.000, E1   +22.266, E3 +588324.761}
SPL {X  -162.820, Y  +531.757, Z    +0.000, E1   +22.276, E3 +588343.816}
SPL {X  -162.820, Y  +527.980, Z    +0.000, E1   +22.326, E3 +588362.647}
SPL {X  -162.820, Y  +524.599, Z    +0.000, E1   +22.287, E3 +588380.044}
SPL {X  -162.820, Y  +522.011, Z    +0.000, E1   +22.282, E3 +588393.121}
SPL {X  -162.820, Y  +519.457, Z    +0.000, E1   +22.481, E3 +588404.410}
SPL {X  -162.820, Y  +505.859, Z    +0.000, E1   +28.367, E3 +588418.893}
SPL {X  -162.820, Y  +504.131, Z    +0.000, E1   +27.325, E3 +588433.032}
SPL {X  -162.820, Y  +503.215, Z    +0.000, E1   +26.369, E3 +588443.718}
SPL {X  -162.820, Y  +502.265, Z    +0.000, E1   +25.287, E3 +588456.200}
SPL {X  -162.820, Y  +501.060, Z    +0.000, E1   +24.081, E3 +588470.940}
SPL {X  -162.820, Y  +500.336, Z    +0.000, E1   +23.110, E3 +588482.080}
SPL {X  -162.820, Y  +499.240, Z    +0.000, E1   +22.316, E3 +588494.391}
SPL {X  -162.820, Y  +498.027, Z    +0.000, E1   +21.516, E3 +588507.298}
SPL {X  -162.820, Y  +495.897, Z    +0.000, E1   +21.662, E3 +588517.219}
SPL {X  -162.820, Y  +493.717, Z    +0.000, E1   +21.704, E3 +588528.325}
SPL {X  -162.820, Y  +491.396, Z    +0.000, E1   +21.707, E3 +588540.449}
SPL {X  -162.820, Y  +488.560, Z    +0.000, E1   +21.695, E3 +588555.558}
SPL {X  -162.820, Y  +485.661, Z    +0.000, E1   +21.712, E3 +588570.444}
SPL {X  -162.820, Y  +483.668, Z    +0.000, E1   +21.664, E3 +588581.271}
SPL {X  -162.820, Y  +481.739, Z    +0.000, E1   +21.704, E3 +588590.985}
SPL {X  -162.820, Y  +479.894, Z    +0.000, E1   +21.695, E3 +588600.772}
SPL {X  -162.820, Y  +477.685, Z    +0.000, E1   +21.656, E3 +588612.710}
SPL {X  -162.820, Y  +475.419, Z    +0.000, E1   +21.711, E3 +588624.062}
SPL {X  -162.820, Y  +473.301, Z    +0.000, E1   +21.712, E3 +588635.160}
SPL {X  -162.820, Y  +470.965, Z    +0.000, E1   +21.700, E3 +588647.504}
SPL {X  -162.820, Y  +469.036, Z    +0.000, E1   +21.695, E3 +588657.548}
SPL {X  -162.820, Y  +467.138, Z    +0.000, E1   +21.678, E3 +588667.720}
SPL {X  -162.820, Y  +465.011, Z    +0.000, E1   +21.692, E3 +588678.702}
SPL {X  -162.820, Y  +462.669, Z    +0.000, E1   +21.752, E3 +588690.483}
SPL {X  -162.820, Y  +460.725, Z    +0.000, E1   +21.689, E3 +588701.096}
SPL {X  -162.820, Y  +458.666, Z    +0.000, E1   +21.695, E3 +588711.908}
SPL {X  -162.820, Y  +456.431, Z    +0.000, E1   +21.708, E3 +588723.436}
SPL {X  -162.820, Y  +453.609, Z    +0.000, E1   +21.757, E3 +588737.970}
SPL {X  -162.820, Y  +450.610, Z    +0.000, E1   +21.698, E3 +588754.028}
SPL {X  -162.820, Y  +448.170, Z    +0.000, E1   +21.667, E3 +588767.048}
SPL {X  -162.820, Y  +445.508, Z    +0.000, E1   +21.732, E3 +588780.567}
SPL {X  -162.820, Y  +442.443, Z    +0.000, E1   +21.712, E3 +588796.687}
SPL {X  -162.820, Y  +439.933, Z    +0.000, E1   +21.690, E3 +588809.968}
SPL {X  -162.820, Y  +437.628, Z    +0.000, E1   +21.678, E3 +588822.156}
SPL {X  -162.820, Y  +434.473, Z    +0.000, E1   +21.747, E3 +588838.253}
SPL {X  -162.820, Y  +431.492, Z    +0.000, E1   +21.686, E3 +588854.201}
SPL {X  -162.820, Y  +429.074, Z    +0.000, E1   +21.710, E3 +588866.653}
SPL {X  -162.820, Y  +426.023, Z    +0.000, E1   +21.718, E3 +588882.721}
SPL {X  -162.820, Y  +422.986, Z    +0.000, E1   +21.685, E3 +588898.768}
SPL {X  -162.820, Y  +420.528, Z    +0.000, E1   +21.706, E3 +588911.418}
SPL {X  -162.820, Y  +418.116, Z    +0.000, E1   +21.761, E3 +588923.566}
SPL {X  -162.820, Y  +416.127, Z    +0.000, E1   +21.715, E3 +588934.271}
SPL {X  -162.820, Y  +414.361, Z    +0.000, E1   +21.613, E3 +588944.458}
SPL {X  -162.820, Y  +411.450, Z    +0.000, E1   +21.710, E3 +588959.032}
SPL {X  -162.820, Y  +408.590, Z    +0.000, E1   +21.735, E3 +588973.657}
SPL {X  -162.820, Y  +406.238, Z    +0.000, E1   +21.697, E3 +588986.306}
SPL {X  -162.820, Y  +403.166, Z    +0.000, E1   +21.746, E3 +589002.112}
SPL {X  -162.820, Y  +400.348, Z    +0.000, E1   +21.713, E3 +589016.947}
SPL {X  -162.820, Y  +398.298, Z    +0.000, E1   +21.721, E3 +589027.562}
SPL {X  -162.820, Y  +396.371, Z    +0.000, E1   +21.713, E3 +589037.744}
SPL {X  -162.820, Y  +394.508, Z    +0.000, E1   +21.616, E3 +589048.300}
SPL {X  -162.820, Y  +391.777, Z    +0.000, E1   +21.714, E3 +589061.959}
SPL {X  -162.820, Y  +388.822, Z    +0.000, E1   +21.717, E3 +589077.279}
SPL {X  -162.820, Y  +386.818, Z    +0.000, E1   +21.679, E3 +589088.019}
SPL {X  -162.820, Y  +384.697, Z    +0.000, E1   +21.693, E3 +589099.089}
SPL {X  -162.820, Y  +382.288, Z    +0.000, E1   +21.742, E3 +589111.212}
SPL {X  -162.817, Y  +379.520, Z    +0.000, E1   +21.723, E3 +589126.050}
SPL {X  -162.776, Y  +376.710, Z    +0.000, E1   +21.698, E3 +589140.789}
SPL {X  -162.707, Y  +374.438, Z    +0.000, E1   +21.688, E3 +589152.793}
SPL {X  -162.607, Y  +372.171, Z    +0.000, E1   +21.692, E3 +589164.592}
SPL {X  -162.494, Y  +370.197, Z    +0.000, E1   +21.655, E3 +589175.219}
SPL {X  -162.349, Y  +368.131, Z    +0.000, E1   +21.624, E3 +589186.337}
SPL {X  -162.161, Y  +365.866, Z    +0.000, E1   +21.642, E3 +589198.022}
SPL {X  -161.927, Y  +363.466, Z    +0.000, E1   +21.730, E3 +589209.793}
SPL {X  -160.290, Y  +351.907, Z    +0.000, E1   +27.562, E3 +589217.371}
SPL {X  -160.281, Y  +351.857, Z    +0.000, E1   +24.243, E3 +589246.784}
ENDSPLINE

SPLINE
SPL {X  -161.833, Y  +362.603, Z    +0.000, E1   +17.021, E3 +589261.480}
ENDSPLINE

SPLINE
SPL {X  -160.786, Y  +354.842, Z    +0.000, E1   +19.274, E3 +589293.636}
ENDSPLINE

SPLINE
SPL {X  -162.485, Y  +370.062, Z    +0.000, E1   +10.606, E3 +589300.014}
SPL {X  -162.820, Y  +381.311, Z    +0.000, E1    +4.054, E3 +589290.369}
SPL {X  -162.820, Y  +390.142, Z    +0.000, E1    -2.185, E3 +589290.697}
SPL {X  -162.820, Y  +393.415, Z    +0.000, E1    -4.587, E3 +589295.805}
SPL {X  -162.820, Y  +399.630, Z    +0.000, E1    -9.426, E3 +589297.734}
SPL {X  -162.820, Y  +408.127, Z    +0.000, E1   -18.417, E3 +589284.023}
SPL {X  -162.820, Y  +420.083, Z    +0.000, E1   -24.325, E3 +589304.498}
SPL {X  -162.820, Y  +428.527, Z    +0.000, E1   -26.988, E3 +589321.790}
SPL {X  -162.820, Y  +431.336, Z    +0.000, E1   -24.162, E3 +589352.000}
SPL {X  -162.820, Y  +432.048, Z    +0.000, E1   -22.832, E3 +589366.504}
SPL {X  -162.820, Y  +434.888, Z    +0.000, E1   -22.823, E3 +589380.453}
SPL {X  -162.820, Y  +436.834, Z    +0.000, E1   -22.779, E3 +589390.413}
SPL {X  -162.820, Y  +438.868, Z    +0.000, E1   -22.837, E3 +589400.067}
SPL {X  -162.820, Y  +441.351, Z    +0.000, E1   -22.805, E3 +589412.642}
SPL {X  -162.820, Y  +443.809, Z    +0.000, E1   -22.804, E3 +589424.809}
SPL {X  -162.820, Y  +447.077, Z    +0.000, E1   -22.869, E3 +589440.619}
SPL {X  -162.820, Y  +449.911, Z    +0.000, E1   -22.774, E3 +589455.229}
SPL {X  -162.820, Y  +451.861, Z    +0.000, E1   -22.750, E3 +589465.076}
SPL {X  -162.820, Y  +454.167, Z    +0.000, E1   -22.842, E3 +589475.805}
SPL {X  -162.820, Y  +456.529, Z    +0.000, E1   -22.855, E3 +589487.334}
SPL {X  -162.820, Y  +458.725, Z    +0.000, E1   -22.793, E3 +589498.738}
SPL {X  -162.820, Y  +461.700, Z    +0.000, E1   -22.822, E3 +589513.361}
SPL {X  -162.820, Y  +464.633, Z    +0.000, E1   -22.813, E3 +589527.858}
SPL {X  -162.820, Y  +466.699, Z    +0.000, E1   -22.824, E3 +589537.904}
SPL {X  -162.820, Y  +468.655, Z    +0.000, E1   -22.858, E3 +589547.347}
SPL {X  -162.820, Y  +470.892, Z    +0.000, E1   -22.837, E3 +589558.586}
SPL {X  -162.820, Y  +473.485, Z    +0.000, E1   -22.806, E3 +589571.784}
SPL {X  -162.820, Y  +475.738, Z    +0.000, E1   -22.728, E3 +589583.449}
SPL {X  -162.820, Y  +478.177, Z    +0.000, E1   -22.834, E3 +589594.789}
SPL {X  -162.820, Y  +481.034, Z    +0.000, E1   -22.831, E3 +589608.926}
SPL {X  -162.820, Y  +483.391, Z    +0.000, E1   -22.793, E3 +589620.862}
SPL {X  -162.820, Y  +486.307, Z    +0.000, E1   -22.833, E3 +589635.116}
SPL {X  -162.820, Y  +489.750, Z    +0.000, E1   -22.832, E3 +589652.187}
SPL {X  -162.820, Y  +492.546, Z    +0.000, E1   -22.823, E3 +589665.945}
SPL {X  -162.820, Y  +495.526, Z    +0.000, E1   -22.833, E3 +589680.827}
SPL {X  -162.820, Y  +499.330, Z    +0.000, E1   -22.841, E3 +589699.609}
SPL {X  -162.820, Y  +503.049, Z    +0.000, E1   -22.823, E3 +589718.158}
SPL {X  -162.820, Y  +506.908, Z    +0.000, E1   -22.877, E3 +589736.828}
SPL {X  -162.820, Y  +510.068, Z    +0.000, E1   -22.761, E3 +589753.299}
SPL {X  -162.820, Y  +512.359, Z    +0.000, E1   -22.823, E3 +589764.031}
SPL {X  -162.820, Y  +513.873, Z    +0.000, E1   -22.800, E3 +589771.718}
SPL {X  -162.820, Y  +516.100, Z    +0.000, E1   -22.809, E3 +589782.794}
SPL {X  -162.820, Y  +518.662, Z    +0.000, E1   -22.847, E3 +589795.093}
SPL {X  -162.820, Y  +520.641, Z    +0.000, E1   -22.790, E3 +589805.334}
SPL {X  -162.820, Y  +523.535, Z    +0.000, E1   -22.857, E3 +589819.303}
SPL {X  -162.820, Y  +526.661, Z    +0.000, E1   -22.801, E3 +589835.127}
SPL {X  -162.820, Y  +528.725, Z    +0.000, E1   -22.770, E3 +589845.496}
SPL {X  -162.820, Y  +530.303, Z    +0.000, E1   -22.798, E3 +589853.115}
SPL {X  -162.820, Y  +532.614, Z    +0.000, E1   -22.828, E3 +589864.384}
SPL {X  -162.820, Y  +534.838, Z    +0.000, E1   -22.864, E3 +589875.012}
SPL {X  -162.820, Y  +536.882, Z    +0.000, E1   -22.782, E3 +589885.867}
SPL {X  -162.820, Y  +539.194, Z    +0.000, E1   -22.826, E3 +589896.916}
SPL {X  -162.820, Y  +541.555, Z    +0.000, E1   -22.817, E3 +589908.730}
SPL {X  -162.820, Y  +543.728, Z    +0.000, E1   -22.799, E3 +589919.588}
SPL {X  -162.820, Y  +545.925, Z    +0.000, E1   -22.803, E3 +589930.458}
SPL {X  -162.820, Y  +549.071, Z    +0.000, E1   -22.836, E3 +589945.985}
SPL {X  -162.820, Y  +553.089, Z    +0.000, E1   -22.838, E3 +589965.885}
SPL {X  -162.820, Y  +556.430, Z    +0.000, E1   -22.821, E3 +589982.386}
SPL {X  -162.820, Y  +559.675, Z    +0.000, E1   -22.837, E3 +589998.466}
SPL {X  -162.820, Y  +562.799, Z    +0.000, E1   -22.814, E3 +590013.973}
SPL {X  -162.820, Y  +565.170, Z    +0.000, E1   -22.801, E3 +590025.797}
SPL {X  -162.820, Y  +568.020, Z    +0.000, E1   -22.787, E3 +590040.184}
SPL {X  -162.820, Y  +570.992, Z    +0.000, E1   -22.834, E3 +590054.403}
SPL {X  -162.820, Y  +572.901, Z    +0.000, E1   -22.775, E3 +590064.272}
SPL {X  -162.820, Y  +575.638, Z    +0.000, E1   -22.855, E3 +590077.381}
SPL {X  -162.820, Y  +578.553, Z    +0.000, E1   -22.801, E3 +590092.093}
SPL {X  -162.820, Y  +581.064, Z    +0.000, E1   -22.823, E3 +590104.378}
SPL {X  -162.820, Y  +583.435, Z    +0.000, E1   -22.808, E3 +590116.200}
SPL {X  -162.820, Y  +585.410, Z    +0.000, E1   -22.764, E3 +590126.335}
SPL {X  -162.820, Y  +587.676, Z    +0.000, E1   -22.853, E3 +590136.850}
SPL {X  -162.820, Y  +589.682, Z    +0.000, E1   -22.776, E3 +590147.380}
SPL {X  -162.820, Y  +591.720, Z    +0.000, E1   -22.868, E3 +590156.691}
SPL {X  -162.820, Y  +593.650, Z    +0.000, E1   -22.810, E3 +590166.760}
SPL {X  -162.820, Y  +595.830, Z    +0.000, E1   -22.828, E3 +590177.376}
SPL {X  -162.820, Y  +598.094, Z    +0.000, E1   -22.843, E3 +590188.489}
SPL {X  -162.820, Y  +600.420, Z    +0.000, E1   -22.826, E3 +590200.121}
SPL {X  -162.820, Y  +602.573, Z    +0.000, E1   -22.830, E3 +590210.706}
SPL {X  -162.820, Y  +604.828, Z    +0.000, E1   -22.784, E3 +590222.344}
SPL {X  -162.820, Y  +608.133, Z    +0.000, E1   -22.831, E3 +590238.462}
SPL {X  -162.820, Y  +611.103, Z    +0.000, E1   -22.785, E3 +590253.388}
SPL {X  -162.820, Y  +613.294, Z    +0.000, E1   -22.780, E3 +590264.261}
SPL {X  -162.820, Y  +615.356, Z    +0.000, E1   -22.799, E3 +590274.318}
SPL {X  -162.820, Y  +617.439, Z    +0.000, E1   -22.808, E3 +590284.576}
SPL {X  -162.820, Y  +619.665, Z    +0.000, E1   -22.817, E3 +590295.544}
SPL {X  -162.820, Y  +621.733, Z    +0.000, E1   -22.759, E3 +590306.268}
SPL {X  -162.820, Y  +624.076, Z    +0.000, E1   -22.774, E3 +590317.774}
SPL {X  -162.820, Y  +627.244, Z    +0.000, E1   -22.803, E3 +590333.456}
SPL {X  -162.820, Y  +630.349, Z    +0.000, E1   -22.766, E3 +590348.988}
SPL {X  -162.820, Y  +632.572, Z    +0.000, E1   -22.785, E3 +590359.794}
SPL {X  -162.820, Y  +634.507, Z    +0.000, E1   -22.784, E3 +590369.433}
SPL {X  -162.820, Y  +636.863, Z    +0.000, E1   -22.760, E3 +590381.355}
SPL {X  -162.820, Y  +640.111, Z    +0.000, E1   -22.809, E3 +590397.238}
SPL {X  -162.820, Y  +643.449, Z    +0.000, E1   -22.796, E3 +590413.756}
SPL {X  -162.820, Y  +645.630, Z    +0.000, E1   -22.795, E3 +590424.452}
SPL {X  -162.820, Y  +647.561, Z    +0.000, E1   -22.705, E3 +590434.903}
SPL {X  -162.820, Y  +649.758, Z    +0.000, E1   -22.780, E3 +590445.093}
SPL {X  -162.820, Y  +651.708, Z    +0.000, E1   -22.810, E3 +590454.587}
SPL {X  -162.820, Y  +653.898, Z    +0.000, E1   -22.796, E3 +590465.508}
SPL {X  -162.820, Y  +656.161, Z    +0.000, E1   -22.812, E3 +590476.629}
SPL {X  -162.820, Y  +658.384, Z    +0.000, E1   -22.822, E3 +590487.496}
SPL {X  -162.820, Y  +660.215, Z    +0.000, E1   -22.649, E3 +590498.086}
SPL {X  -162.820, Y  +662.823, Z    +0.000, E1   -22.799, E3 +590509.794}
SPL {X  -162.820, Y  +665.112, Z    +0.000, E1   -22.835, E3 +590520.849}
SPL {X  -162.820, Y  +667.016, Z    +0.000, E1   -22.823, E3 +590530.277}
SPL {X  -162.820, Y  +668.960, Z    +0.000, E1   -22.773, E3 +590540.445}
SPL {X  -162.820, Y  +672.333, Z    +0.000, E1   -22.837, E3 +590556.781}
SPL {X  -162.812, Y  +675.071, Z    +0.000, E1   -22.742, E3 +590570.926}
SPL {X  -162.773, Y  +677.428, Z    +0.000, E1   -22.762, E3 +590582.523}
SPL {X  -162.691, Y  +679.987, Z    +0.000, E1   -22.794, E3 +590594.936}
SPL {X  -162.604, Y  +681.880, Z    +0.000, E1   -22.691, E3 +590605.097}
SPL {X  -162.458, Y  +684.346, Z    +0.000, E1   -22.764, E3 +590616.891}
SPL {X  -162.296, Y  +686.547, Z    +0.000, E1   -22.660, E3 +590628.508}
SPL {X  -162.090, Y  +688.902, Z    +0.000, E1   -22.700, E3 +590640.016}
SPL {X  -161.474, Y  +694.390, Z    +0.000, E1   -24.298, E3 +590653.371}
SPL {X  -158.730, Y  +709.763, Z    +0.000, E1   -31.225, E3 +590664.710}
ENDSPLINE

SPLINE
SPL {X  -160.932, Y  +698.225, Z    +0.000, E1   -21.712, E3 +590695.819}
SPL {X  -161.691, Y  +692.643, Z    +0.000, E1   -17.369, E3 +590712.702}
SPL {X  -162.534, Y  +683.153, Z    +0.000, E1   -10.475, E3 +590738.169}
SPL {X  -162.820, Y  +667.630, Z    +0.000, E1    -0.882, E3 +590732.145}
SPL {X  -162.820, Y  +661.883, Z    +0.000, E1    +3.373, E3 +590737.588}
SPL {X  -162.820, Y  +653.808, Z    +0.000, E1    +9.891, E3 +590735.280}
SPL {X  -162.820, Y  +632.548, Z    +0.000, E1   +27.446, E3 +590731.816}
ENDSPLINE

SPLINE
SPL {X  -162.820, Y  +638.080, Z    +0.000, E1   +18.858, E3 +590759.565}
ENDSPLINE

SPLINE
SPL {X  -162.820, Y  +623.278, Z    +0.000, E1   +28.723, E3 +590761.135}
SPL {X  -162.820, Y  +618.658, Z    +0.000, E1   +26.841, E3 +590789.744}
ENDSPLINE

SPLINE
SPL {X  -162.820, Y  +623.685, Z    +0.000, E1   +22.346, E3 +590802.051}
ENDSPLINE

SPLINE
SPL {X  -162.820, Y  +621.304, Z    +0.000, E1   +22.259, E3 +590814.866}
SPL {X  -162.820, Y  +618.758, Z    +0.000, E1   +22.239, E3 +590828.017}
SPL {X  -162.820, Y  +616.062, Z    +0.000, E1   +22.275, E3 +590841.438}
SPL {X  -162.820, Y  +613.536, Z    +0.000, E1   +22.242, E3 +590854.559}
SPL {X  -162.820, Y  +611.128, Z    +0.000, E1   +22.252, E3 +590866.730}
SPL {X  -162.820, Y  +608.428, Z    +0.000, E1   +22.255, E3 +590880.513}
SPL {X  -162.820, Y  +605.178, Z    +0.000, E1   +22.267, E3 +590897.045}
SPL {X  -162.820, Y  +602.350, Z    +0.000, E1   +22.224, E3 +590911.663}
SPL {X  -162.820, Y  +599.842, Z    +0.000, E1   +22.298, E3 +590923.814}
SPL {X  -162.820, Y  +597.194, Z    +0.000, E1   +22.253, E3 +590937.735}
SPL {X  -162.820, Y  +594.779, Z    +0.000, E1   +22.284, E3 +590949.639}
SPL {X  -162.820, Y  +592.389, Z    +0.000, E1   +22.245, E3 +590962.256}
SPL {X  -162.820, Y  +589.492, Z    +0.000, E1   +22.304, E3 +590976.440}
SPL {X  -162.820, Y  +587.447, Z    +0.000, E1   +22.279, E3 +590986.969}
SPL {X  -162.820, Y  +585.192, Z    +0.000, E1   +22.298, E3 +590998.379}
SPL {X  -162.820, Y  +582.610, Z    +0.000, E1   +22.234, E3 +591012.002}
SPL {X  -162.820, Y  +580.317, Z    +0.000, E1   +22.300, E3 +591023.056}
SPL {X  -162.820, Y  +578.878, Z    +0.000, E1   +22.272, E3 +591030.566}
SPL {X  -162.820, Y  +576.856, Z    +0.000, E1   +22.233, E3 +591041.324}
SPL {X  -162.820, Y  +574.811, Z    +0.000, E1   +22.236, E3 +591051.588}
SPL {X  -162.820, Y  +572.645, Z    +0.000, E1   +22.246, E3 +591062.683}
SPL {X  -162.820, Y  +569.475, Z    +0.000, E1   +22.269, E3 +591078.689}
SPL {X  -162.820, Y  +565.838, Z    +0.000, E1   +22.271, E3 +591097.284}
SPL {X  -162.820, Y  +562.162, Z    +0.000, E1   +22.252, E3 +591116.101}
SPL {X  -162.820, Y  +558.919, Z    +0.000, E1   +22.286, E3 +591132.265}
SPL {X  -162.820, Y  +556.169, Z    +0.000, E1   +22.295, E3 +591146.094}
SPL {X  -162.820, Y  +553.294, Z    +0.000, E1   +22.266, E3 +591161.092}
SPL {X  -162.820, Y  +550.136, Z    +0.000, E1   +22.258, E3 +591177.205}
SPL {X  -162.820, Y  +546.694, Z    +0.000, E1   +22.290, E3 +591194.527}
SPL {X  -162.820, Y  +543.558, Z    +0.000, E1   +22.285, E3 +591210.390}
SPL {X  -162.820, Y  +541.633, Z    +0.000, E1   +22.257, E3 +591220.318}
SPL {X  -162.820, Y  +539.116, Z    +0.000, E1   +22.302, E3 +591232.929}
SPL {X  -162.820, Y  +536.913, Z    +0.000, E1   +22.192, E3 +591244.853}
SPL {X  -162.820, Y  +534.880, Z    +0.000, E1   +22.252, E3 +591254.807}
SPL {X  -162.820, Y  +532.896, Z    +0.000, E1   +22.234, E3 +591264.967}
SPL {X  -162.820, Y  +531.056, Z    +0.000, E1   +22.251, E3 +591274.249}
SPL {X  -162.820, Y  +528.708, Z    +0.000, E1   +22.319, E3 +591285.631}
SPL {X  -162.820, Y  +525.932, Z    +0.000, E1   +22.258, E3 +591300.387}
SPL {X  -162.820, Y  +522.524, Z    +0.000, E1   +22.326, E3 +591317.111}
SPL {X  -162.820, Y  +519.457, Z    +0.000, E1   +22.481, E3 +591331.240}
SPL {X  -162.820, Y  +506.285, Z    +0.000, E1   +28.538, E3 +591342.697}
SPL {X  -162.820, Y  +504.441, Z    +0.000, E1   +27.574, E3 +591357.040}
SPL {X  -162.820, Y  +502.813, Z    +0.000, E1   +26.013, E3 +591375.237}
SPL {X  -162.820, Y  +502.016, Z    +0.000, E1   +24.802, E3 +591387.580}
SPL {X  -162.820, Y  +501.060, Z    +0.000, E1   +24.081, E3 +591397.769}
SPL {X  -162.820, Y  +499.934, Z    +0.000, E1   +22.814, E3 +591413.638}
SPL {X  -162.820, Y  +498.303, Z    +0.000, E1   +21.749, E3 +591430.894}
SPL {X  -162.820, Y  +495.897, Z    +0.000, E1   +21.662, E3 +591444.048}
SPL {X  -162.820, Y  +493.717, Z    +0.000, E1   +21.704, E3 +591455.154}
SPL {X  -162.820, Y  +491.396, Z    +0.000, E1   +21.707, E3 +591467.278}
SPL {X  -162.820, Y  +489.485, Z    +0.000, E1   +21.661, E3 +591477.626}
SPL {X  -162.820, Y  +487.723, Z    +0.000, E1   +21.665, E3 +591486.829}
SPL {X  -162.820, Y  +485.661, Z    +0.000, E1   +21.712, E3 +591497.273}
SPL {X  -162.820, Y  +482.775, Z    +0.000, E1   +21.716, E3 +591512.525}
SPL {X  -162.820, Y  +479.894, Z    +0.000, E1   +21.695, E3 +591527.601}
SPL {X  -162.820, Y  +477.685, Z    +0.000, E1   +21.656, E3 +591539.539}
SPL {X  -162.820, Y  +475.419, Z    +0.000, E1   +21.711, E3 +591550.892}
SPL {X  -162.820, Y  +473.301, Z    +0.000, E1   +21.712, E3 +591561.989}
SPL {X  -162.820, Y  +470.965, Z    +0.000, E1   +21.700, E3 +591574.334}
SPL {X  -162.820, Y  +469.036, Z    +0.000, E1   +21.695, E3 +591584.378}
SPL {X  -162.820, Y  +467.138, Z    +0.000, E1   +21.678, E3 +591594.549}
SPL {X  -162.820, Y  +465.011, Z    +0.000, E1   +21.692, E3 +591605.532}
SPL {X  -162.820, Y  +462.669, Z    +0.000, E1   +21.752, E3 +591617.312}
SPL {X  -162.820, Y  +460.725, Z    +0.000, E1   +21.689, E3 +591627.925}
SPL {X  -162.820, Y  +458.666, Z    +0.000, E1   +21.695, E3 +591638.737}
SPL {X  -162.820, Y  +456.431, Z    +0.000, E1   +21.708, E3 +591650.266}
SPL {X  -162.820, Y  +454.628, Z    +0.000, E1   +21.674, E3 +591659.984}
SPL {X  -162.820, Y  +452.690, Z    +0.000, E1   +21.773, E3 +591669.258}
SPL {X  -162.820, Y  +450.610, Z    +0.000, E1   +21.698, E3 +591680.857}
SPL {X  -162.820, Y  +448.170, Z    +0.000, E1   +21.667, E3 +591693.878}
SPL {X  -162.820, Y  +446.246, Z    +0.000, E1   +21.696, E3 +591703.695}
SPL {X  -162.820, Y  +443.784, Z    +0.000, E1   +21.713, E3 +591716.482}
SPL {X  -162.820, Y  +440.567, Z    +0.000, E1   +21.731, E3 +591733.321}
SPL {X  -162.820, Y  +437.628, Z    +0.000, E1   +21.678, E3 +591748.985}
SPL {X  -162.820, Y  +435.262, Z    +0.000, E1   +21.727, E3 +591760.921}
SPL {X  -162.820, Y  +433.510, Z    +0.000, E1   +21.692, E3 +591770.335}
SPL {X  -162.820, Y  +431.492, Z    +0.000, E1   +21.686, E3 +591781.030}
SPL {X  -162.820, Y  +429.074, Z    +0.000, E1   +21.710, E3 +591793.482}
SPL {X  -162.820, Y  +427.020, Z    +0.000, E1   +21.674, E3 +591804.484}
SPL {X  -162.820, Y  +424.525, Z    +0.000, E1   +21.712, E3 +591817.397}
SPL {X  -162.820, Y  +421.144, Z    +0.000, E1   +21.719, E3 +591835.064}
SPL {X  -162.820, Y  +418.116, Z    +0.000, E1   +21.761, E3 +591850.395}
SPL {X  -162.820, Y  +416.127, Z    +0.000, E1   +21.715, E3 +591861.100}
SPL {X  -162.820, Y  +414.361, Z    +0.000, E1   +21.613, E3 +591871.287}
SPL {X  -162.820, Y  +412.134, Z    +0.000, E1   +21.697, E3 +591882.232}
SPL {X  -162.820, Y  +409.248, Z    +0.000, E1   +21.741, E3 +591897.167}
SPL {X  -162.820, Y  +406.238, Z    +0.000, E1   +21.697, E3 +591913.135}
SPL {X  -162.820, Y  +404.001, Z    +0.000, E1   +21.723, E3 +591924.565}
SPL {X  -162.820, Y  +402.223, Z    +0.000, E1   +21.697, E3 +591934.050}
SPL {X  -162.820, Y  +400.348, Z    +0.000, E1   +21.713, E3 +591943.776}
SPL {X  -162.820, Y  +398.298, Z    +0.000, E1   +21.721, E3 +591954.392}
SPL {X  -162.820, Y  +396.371, Z    +0.000, E1   +21.713, E3 +591964.573}
SPL {X  -162.820, Y  +394.508, Z    +0.000, E1   +21.616, E3 +591975.129}
SPL {X  -162.820, Y  +392.435, Z    +0.000, E1   +21.681, E3 +591985.482}
SPL {X  -162.820, Y  +389.390, Z    +0.000, E1   +21.742, E3 +592001.089}
SPL {X  -162.820, Y  +386.818, Z    +0.000, E1   +21.679, E3 +592014.848}
SPL {X  -162.820, Y  +384.697, Z    +0.000, E1   +21.693, E3 +592025.918}
SPL {X  -162.820, Y  +382.288, Z    +0.000, E1   +21.742, E3 +592038.042}
SPL {X  -162.817, Y  +379.520, Z    +0.000, E1   +21.723, E3 +592052.879}
SPL {X  -162.776, Y  +376.710, Z    +0.000, E1   +21.698, E3 +592067.618}
SPL {X  -162.707, Y  +374.438, Z    +0.000, E1   +21.688, E3 +592079.622}
SPL {X  -162.607, Y  +372.171, Z    +0.000, E1   +21.692, E3 +592091.422}
SPL {X  -162.494, Y  +370.197, Z    +0.000, E1   +21.655, E3 +592102.048}
SPL {X  -162.349, Y  +368.131, Z    +0.000, E1   +21.624, E3 +592113.166}
SPL {X  -162.161, Y  +365.866, Z    +0.000, E1   +21.642, E3 +592124.851}
SPL {X  -161.651, Y  +361.024, Z    +0.000, E1   +22.970, E3 +592138.274}
SPL {X  -160.281, Y  +351.857, Z    +0.000, E1   +24.243, E3 +592173.614}
ENDSPLINE

SPLINE
SPL {X  -161.833, Y  +362.603, Z    +0.000, E1   +17.021, E3 +592188.309}
ENDSPLINE

SPLINE
SPL {X  -160.786, Y  +354.842, Z    +0.000, E1   +19.274, E3 +592220.465}
ENDSPLINE

SPLINE
SPL {X  -162.485, Y  +370.062, Z    +0.000, E1   +10.606, E3 +592226.843}
SPL {X  -162.818, Y  +379.636, Z    +0.000, E1    +5.115, E3 +592216.192}
SPL {X  -162.820, Y  +386.976, Z    +0.000, E1    +0.144, E3 +592215.291}
SPL {X  -162.820, Y  +391.982, Z    +0.000, E1    -3.443, E3 +592222.056}
SPL {X  -162.820, Y  +399.630, Z    +0.000, E1    -9.426, E3 +592224.563}
SPL {X  -162.820, Y  +408.127, Z    +0.000, E1   -18.417, E3 +592210.852}
SPL {X  -162.820, Y  +420.083, Z    +0.000, E1   -24.325, E3 +592231.327}
SPL {X  -162.820, Y  +428.527, Z    +0.000, E1   -26.988, E3 +592248.619}
SPL {X  -162.820, Y  +431.336, Z    +0.000, E1   -24.162, E3 +592278.829}
SPL {X  -162.820, Y  +432.048, Z    +0.000, E1   -22.832, E3 +592293.333}
SPL {X  -162.820, Y  +434.888, Z    +0.000, E1   -22.823, E3 +592307.283}
SPL {X  -162.820, Y  +436.834, Z    +0.000, E1   -22.779, E3 +592317.243}
SPL {X  -162.820, Y  +438.868, Z    +0.000, E1   -22.837, E3 +592326.896}
SPL {X  -162.820, Y  +441.351, Z    +0.000, E1   -22.805, E3 +592339.472}
SPL {X  -162.820, Y  +443.809, Z    +0.000, E1   -22.804, E3 +592351.638}
SPL {X  -162.820, Y  +447.077, Z    +0.000, E1   -22.869, E3 +592367.448}
SPL {X  -162.820, Y  +449.911, Z    +0.000, E1   -22.774, E3 +592382.058}
SPL {X  -162.820, Y  +451.861, Z    +0.000, E1   -22.750, E3 +592391.905}
SPL {X  -162.820, Y  +454.167, Z    +0.000, E1   -22.842, E3 +592402.635}
SPL {X  -162.820, Y  +456.529, Z    +0.000, E1   -22.855, E3 +592414.163}
SPL {X  -162.820, Y  +458.725, Z    +0.000, E1   -22.793, E3 +592425.568}
SPL {X  -162.820, Y  +461.700, Z    +0.000, E1   -22.822, E3 +592440.190}
SPL {X  -162.820, Y  +464.633, Z    +0.000, E1   -22.813, E3 +592454.687}
SPL {X  -162.820, Y  +467.913, Z    +0.000, E1   -22.879, E3 +592470.526}
SPL {X  -162.820, Y  +470.892, Z    +0.000, E1   -22.837, E3 +592485.415}
SPL {X  -162.820, Y  +472.726, Z    +0.000, E1   -22.777, E3 +592494.954}
SPL {X  -162.820, Y  +475.118, Z    +0.000, E1   -22.777, E3 +592506.925}
SPL {X  -162.820, Y  +477.389, Z    +0.000, E1   -22.803, E3 +592517.842}
SPL {X  -162.820, Y  +478.914, Z    +0.000, E1   -22.821, E3 +592525.234}
SPL {X  -162.820, Y  +481.034, Z    +0.000, E1   -22.831, E3 +592535.756}
SPL {X  -162.820, Y  +484.256, Z    +0.000, E1   -22.840, E3 +592551.774}
SPL {X  -162.820, Y  +487.952, Z    +0.000, E1   -22.824, E3 +592570.205}
SPL {X  -162.820, Y  +491.768, Z    +0.000, E1   -22.852, E3 +592588.885}
SPL {X  -162.820, Y  +495.526, Z    +0.000, E1   -22.833, E3 +592607.657}
SPL {X  -162.820, Y  +499.330, Z    +0.000, E1   -22.841, E3 +592626.438}
SPL {X  -162.820, Y  +502.361, Z    +0.000, E1   -22.801, E3 +592641.596}
SPL {X  -162.820, Y  +505.323, Z    +0.000, E1   -22.838, E3 +592656.068}
SPL {X  -162.820, Y  +508.611, Z    +0.000, E1   -22.838, E3 +592672.331}
SPL {X  -162.820, Y  +511.620, Z    +0.000, E1   -22.791, E3 +592687.575}
SPL {X  -162.820, Y  +513.873, Z    +0.000, E1   -22.800, E3 +592698.547}
SPL {X  -162.820, Y  +516.100, Z    +0.000, E1   -22.809, E3 +592709.623}
SPL {X  -162.820, Y  +518.662, Z    +0.000, E1   -22.847, E3 +592721.922}
SPL {X  -162.820, Y  +520.641, Z    +0.000, E1   -22.790, E3 +592732.163}
SPL {X  -162.820, Y  +522.740, Z    +0.000, E1   -22.811, E3 +592742.405}
SPL {X  -162.820, Y  +524.628, Z    +0.000, E1   -22.846, E3 +592751.401}
SPL {X  -162.820, Y  +526.661, Z    +0.000, E1   -22.801, E3 +592761.956}
SPL {X  -162.820, Y  +529.662, Z    +0.000, E1   -22.810, E3 +592776.807}
SPL {X  -162.820, Y  +532.614, Z    +0.000, E1   -22.828, E3 +592791.213}
SPL {X  -162.820, Y  +534.838, Z    +0.000, E1   -22.864, E3 +592801.842}
SPL {X  -162.820, Y  +536.882, Z    +0.000, E1   -22.782, E3 +592812.697}
SPL {X  -162.820, Y  +539.194, Z    +0.000, E1   -22.826, E3 +592823.745}
SPL {X  -162.820, Y  +541.555, Z    +0.000, E1   -22.817, E3 +592835.560}
SPL {X  -162.820, Y  +543.728, Z    +0.000, E1   -22.799, E3 +592846.417}
SPL {X  -162.820, Y  +545.925, Z    +0.000, E1   -22.803, E3 +592857.287}
SPL {X  -162.820, Y  +549.071, Z    +0.000, E1   -22.836, E3 +592872.814}
SPL {X  -162.820, Y  +553.089, Z    +0.000, E1   -22.838, E3 +592892.714}
SPL {X  -162.820, Y  +556.430, Z    +0.000, E1   -22.821, E3 +592909.215}
SPL {X  -162.820, Y  +558.974, Z    +0.000, E1   -22.806, E3 +592921.915}
SPL {X  -162.820, Y  +562.171, Z    +0.000, E1   -22.845, E3 +592937.613}
SPL {X  -162.820, Y  +565.170, Z    +0.000, E1   -22.801, E3 +592952.627}
SPL {X  -162.820, Y  +567.308, Z    +0.000, E1   -22.750, E3 +592963.643}
SPL {X  -162.820, Y  +570.378, Z    +0.000, E1   -22.843, E3 +592978.267}
SPL {X  -162.820, Y  +573.634, Z    +0.000, E1   -22.827, E3 +592994.411}
SPL {X  -162.820, Y  +576.228, Z    +0.000, E1   -22.814, E3 +593007.307}
SPL {X  -162.820, Y  +578.553, Z    +0.000, E1   -22.801, E3 +593018.923}
SPL {X  -162.820, Y  +581.064, Z    +0.000, E1   -22.823, E3 +593031.207}
SPL {X  -162.820, Y  +583.435, Z    +0.000, E1   -22.808, E3 +593043.029}
SPL {X  -162.820, Y  +585.410, Z    +0.000, E1   -22.764, E3 +593053.165}
SPL {X  -162.820, Y  +587.676, Z    +0.000, E1   -22.853, E3 +593063.679}
SPL {X  -162.820, Y  +589.682, Z    +0.000, E1   -22.776, E3 +593074.209}
SPL {X  -162.820, Y  +591.720, Z    +0.000, E1   -22.868, E3 +593083.520}
SPL {X  -162.820, Y  +593.650, Z    +0.000, E1   -22.810, E3 +593093.590}
SPL {X  -162.820, Y  +595.830, Z    +0.000, E1   -22.828, E3 +593104.206}
SPL {X  -162.820, Y  +598.094, Z    +0.000, E1   -22.843, E3 +593115.319}
SPL {X  -162.820, Y  +600.420, Z    +0.000, E1   -22.826, E3 +593126.950}
SPL {X  -162.820, Y  +602.573, Z    +0.000, E1   -22.830, E3 +593137.535}
SPL {X  -162.820, Y  +604.828, Z    +0.000, E1   -22.784, E3 +593149.173}
SPL {X  -162.820, Y  +608.133, Z    +0.000, E1   -22.831, E3 +593165.291}
SPL {X  -162.820, Y  +611.103, Z    +0.000, E1   -22.785, E3 +593180.217}
SPL {X  -162.820, Y  +613.294, Z    +0.000, E1   -22.780, E3 +593191.090}
SPL {X  -162.820, Y  +615.356, Z    +0.000, E1   -22.799, E3 +593201.147}
SPL {X  -162.820, Y  +617.439, Z    +0.000, E1   -22.808, E3 +593211.406}
SPL {X  -162.820, Y  +619.665, Z    +0.000, E1   -22.817, E3 +593222.374}
SPL {X  -162.820, Y  +621.733, Z    +0.000, E1   -22.759, E3 +593233.098}
SPL {X  -162.820, Y  +624.076, Z    +0.000, E1   -22.774, E3 +593244.603}
SPL {X  -162.820, Y  +627.244, Z    +0.000, E1   -22.803, E3 +593260.285}
SPL {X  -162.820, Y  +630.349, Z    +0.000, E1   -22.766, E3 +593275.817}
SPL {X  -162.820, Y  +632.572, Z    +0.000, E1   -22.785, E3 +593286.624}
SPL {X  -162.820, Y  +634.507, Z    +0.000, E1   -22.784, E3 +593296.262}
SPL {X  -162.820, Y  +636.863, Z    +0.000, E1   -22.760, E3 +593308.185}
SPL {X  -162.820, Y  +640.111, Z    +0.000, E1   -22.809, E3 +593324.067}
SPL {X  -162.820, Y  +643.449, Z    +0.000, E1   -22.796, E3 +593340.585}
SPL {X  -162.820, Y  +645.630, Z    +0.000, E1   -22.795, E3 +593351.281}
SPL {X  -162.820, Y  +647.561, Z    +0.000, E1   -22.705, E3 +593361.732}
SPL {X  -162.820, Y  +651.051, Z    +0.000, E1   -22.833, E3 +593378.151}
SPL {X  -162.820, Y  +653.898, Z    +0.000, E1   -22.796, E3 +593392.337}
SPL {X  -162.820, Y  +656.161, Z    +0.000, E1   -22.812, E3 +593403.459}
SPL {X  -162.820, Y  +658.384, Z    +0.000, E1   -22.822, E3 +593414.325}
SPL {X  -162.820, Y  +660.215, Z    +0.000, E1   -22.649, E3 +593424.916}
SPL {X  -162.820, Y  +662.823, Z    +0.000, E1   -22.799, E3 +593436.623}
SPL {X  -162.820, Y  +665.112, Z    +0.000, E1   -22.835, E3 +593447.678}
SPL {X  -162.820, Y  +667.016, Z    +0.000, E1   -22.823, E3 +593457.106}
SPL {X  -162.820, Y  +668.960, Z    +0.000, E1   -22.773, E3 +593467.274}
SPL {X  -162.820, Y  +671.605, Z    +0.000, E1   -22.777, E3 +593480.348}
SPL {X  -162.817, Y  +674.515, Z    +0.000, E1   -22.816, E3 +593494.545}
SPL {X  -162.773, Y  +677.428, Z    +0.000, E1   -22.762, E3 +593509.352}
SPL {X  -162.691, Y  +679.987, Z    +0.000, E1   -22.794, E3 +593521.766}
SPL {X  -162.604, Y  +681.880, Z    +0.000, E1   -22.691, E3 +593531.926}
SPL {X  -162.458, Y  +684.346, Z    +0.000, E1   -22.764, E3 +593543.720}
SPL {X  -162.229, Y  +687.364, Z    +0.000, E1   -22.685, E3 +593559.340}
SPL {X  -161.938, Y  +690.422, Z    +0.000, E1   -22.769, E3 +593573.746}
SPL {X  -161.065, Y  +697.344, Z    +0.000, E1   -25.698, E3 +593582.865}
SPL {X  -158.730, Y  +709.763, Z    +0.000, E1   -31.225, E3 +593591.539}
ENDSPLINE

SPLINE
SPL {X  -160.932, Y  +698.225, Z    +0.000, E1   -21.712, E3 +593622.648}
SPL {X  -161.691, Y  +692.643, Z    +0.000, E1   -17.369, E3 +593639.531}
SPL {X  -162.534, Y  +683.153, Z    +0.000, E1   -10.475, E3 +593664.998}
SPL {X  -162.820, Y  +670.105, Z    +0.000, E1    -2.484, E3 +593657.645}
SPL {X  -162.820, Y  +665.819, Z    +0.000, E1    +0.492, E3 +593659.941}
SPL {X  -162.820, Y  +661.883, Z    +0.000, E1    +3.373, E3 +593664.418}
SPL {X  -162.820, Y  +655.163, Z    +0.000, E1    +8.702, E3 +593664.016}
SPL {X  -162.820, Y  +634.515, Z    +0.000, E1   +26.439, E3 +593656.430}
ENDSPLINE

SPLINE
SPL {X  -162.820, Y  +638.080, Z    +0.000, E1   +18.858, E3 +593686.394}
ENDSPLINE

SPLINE
SPL {X  -162.820, Y  +623.278, Z    +0.000, E1   +28.723, E3 +593687.965}
SPL {X  -162.820, Y  +618.658, Z    +0.000, E1   +26.841, E3 +593716.574}
ENDSPLINE

SPLINE
SPL {X  -162.820, Y  +623.685, Z    +0.000, E1   +22.346, E3 +593728.880}
ENDSPLINE

SPLINE
SPL {X  -162.820, Y  +621.304, Z    +0.000, E1   +22.259, E3 +593741.696}
SPL {X  -162.820, Y  +618.758, Z    +0.000, E1   +22.239, E3 +593754.846}
SPL {X  -162.820, Y  +616.062, Z    +0.000, E1   +22.275, E3 +593768.267}
SPL {X  -162.820, Y  +613.536, Z    +0.000, E1   +22.242, E3 +593781.388}
SPL {X  -162.820, Y  +611.128, Z    +0.000, E1   +22.252, E3 +593793.559}
SPL {X  -162.820, Y  +608.428, Z    +0.000, E1   +22.255, E3 +593807.343}
SPL {X  -162.820, Y  +605.984, Z    +0.000, E1   +22.221, E3 +593819.979}
SPL {X  -162.820, Y  +603.020, Z    +0.000, E1   +22.272, E3 +593834.878}
SPL {X  -162.820, Y  +599.168, Z    +0.000, E1   +22.310, E3 +593854.146}
SPL {X  -162.820, Y  +595.597, Z    +0.000, E1   +22.284, E3 +593872.482}
SPL {X  -162.820, Y  +593.320, Z    +0.000, E1   +22.199, E3 +593884.572}
SPL {X  -162.820, Y  +591.031, Z    +0.000, E1   +22.283, E3 +593895.663}
SPL {X  -162.820, Y  +588.026, Z    +0.000, E1   +22.301, E3 +593910.790}
SPL {X  -162.820, Y  +585.899, Z    +0.000, E1   +22.286, E3 +593921.592}
SPL {X  -162.820, Y  +583.204, Z    +0.000, E1   +22.278, E3 +593935.615}
SPL {X  -162.820, Y  +580.317, Z    +0.000, E1   +22.300, E3 +593949.886}
SPL {X  -162.820, Y  +578.061, Z    +0.000, E1   +22.264, E3 +593961.771}
SPL {X  -162.820, Y  +575.394, Z    +0.000, E1   +22.240, E3 +593975.515}
SPL {X  -162.820, Y  +573.156, Z    +0.000, E1   +22.254, E3 +593986.725}
SPL {X  -162.820, Y  +570.852, Z    +0.000, E1   +22.234, E3 +593998.749}
SPL {X  -162.820, Y  +568.608, Z    +0.000, E1   +22.253, E3 +594009.882}
SPL {X  -162.820, Y  +565.838, Z    +0.000, E1   +22.271, E3 +594024.114}
SPL {X  -162.820, Y  +562.162, Z    +0.000, E1   +22.252, E3 +594042.931}
SPL {X  -162.820, Y  +558.919, Z    +0.000, E1   +22.286, E3 +594059.094}
SPL {X  -162.820, Y  +556.169, Z    +0.000, E1   +22.295, E3 +594072.923}
SPL {X  -162.820, Y  +553.294, Z    +0.000, E1   +22.266, E3 +594087.921}
SPL {X  -162.820, Y  +550.136, Z    +0.000, E1   +22.258, E3 +594104.034}
SPL {X  -162.820, Y  +546.694, Z    +0.000, E1   +22.290, E3 +594121.356}
SPL {X  -162.820, Y  +543.558, Z    +0.000, E1   +22.285, E3 +594137.219}
SPL {X  -162.820, Y  +541.633, Z    +0.000, E1   +22.257, E3 +594147.147}
SPL {X  -162.820, Y  +539.116, Z    +0.000, E1   +22.302, E3 +594159.758}
SPL {X  -162.820, Y  +536.913, Z    +0.000, E1   +22.192, E3 +594171.682}
SPL {X  -162.820, Y  +534.880, Z    +0.000, E1   +22.252, E3 +594181.636}
SPL {X  -162.820, Y  +532.896, Z    +0.000, E1   +22.234, E3 +594191.796}
SPL {X  -162.820, Y  +531.056, Z    +0.000, E1   +22.251, E3 +594201.078}
SPL {X  -162.820, Y  +528.708, Z    +0.000, E1   +22.319, E3 +594212.460}
SPL {X  -162.820, Y  +526.907, Z    +0.000, E1   +22.243, E3 +594222.180}
SPL {X  -162.820, Y  +524.599, Z    +0.000, E1   +22.287, E3 +594233.702}
SPL {X  -162.820, Y  +522.011, Z    +0.000, E1   +22.282, E3 +594246.779}
SPL {X  -162.820, Y  +519.457, Z    +0.000, E1   +22.481, E3 +594258.069}
SPL {X  -162.820, Y  +505.859, Z    +0.000, E1   +28.367, E3 +594272.552}
SPL {X  -162.820, Y  +504.131, Z    +0.000, E1   +27.325, E3 +594286.690}
SPL {X  -162.820, Y  +503.215, Z    +0.000, E1   +26.369, E3 +594297.376}
SPL {X  -162.820, Y  +502.502, Z    +0.000, E1   +25.597, E3 +594306.223}
SPL {X  -162.820, Y  +501.672, Z    +0.000, E1   +24.583, E3 +594317.838}
SPL {X  -162.820, Y  +500.515, Z    +0.000, E1   +23.444, E3 +594332.368}
SPL {X  -162.820, Y  +499.633, Z    +0.000, E1   +22.486, E3 +594344.414}
SPL {X  -162.820, Y  +498.303, Z    +0.000, E1   +21.749, E3 +594357.723}
SPL {X  -162.820, Y  +495.897, Z    +0.000, E1   +21.662, E3 +594370.877}
SPL {X  -162.820, Y  +493.717, Z    +0.000, E1   +21.704, E3 +594381.983}
SPL {X  -162.820, Y  +491.396, Z    +0.000, E1   +21.707, E3 +594394.107}
SPL {X  -162.820, Y  +489.485, Z    +0.000, E1   +21.661, E3 +594404.455}
SPL {X  -162.820, Y  +487.723, Z    +0.000, E1   +21.665, E3 +594413.659}
SPL {X  -162.820, Y  +485.661, Z    +0.000, E1   +21.712, E3 +594424.102}
SPL {X  -162.820, Y  +482.775, Z    +0.000, E1   +21.716, E3 +594439.355}
SPL {X  -162.820, Y  +479.894, Z    +0.000, E1   +21.695, E3 +594454.431}
SPL {X  -162.820, Y  +477.685, Z    +0.000, E1   +21.656, E3 +594466.368}
SPL {X  -162.820, Y  +475.419, Z    +0.000, E1   +21.711, E3 +594477.721}
SPL {X  -162.820, Y  +473.301, Z    +0.000, E1   +21.712, E3 +594488.818}
SPL {X  -162.820, Y  +470.965, Z    +0.000, E1   +21.700, E3 +594501.163}
SPL {X  -162.820, Y  +469.036, Z    +0.000, E1   +21.695, E3 +594511.207}
SPL {X  -162.820, Y  +467.138, Z    +0.000, E1   +21.678, E3 +594521.378}
SPL {X  -162.820, Y  +465.011, Z    +0.000, E1   +21.692, E3 +594532.361}
SPL {X  -162.820, Y  +462.669, Z    +0.000, E1   +21.752, E3 +594544.141}
SPL {X  -162.820, Y  +460.725, Z    +0.000, E1   +21.689, E3 +594554.754}
SPL {X  -162.820, Y  +458.666, Z    +0.000, E1   +21.695, E3 +594565.566}
SPL {X  -162.820, Y  +456.431, Z    +0.000, E1   +21.708, E3 +594577.095}
SPL {X  -162.820, Y  +453.609, Z    +0.000, E1   +21.757, E3 +594591.629}
SPL {X  -162.820, Y  +450.610, Z    +0.000, E1   +21.698, E3 +594607.686}
SPL {X  -162.820, Y  +448.170, Z    +0.000, E1   +21.667, E3 +594620.707}
SPL {X  -162.820, Y  +445.508, Z    +0.000, E1   +21.732, E3 +594634.225}
SPL {X  -162.820, Y  +442.443, Z    +0.000, E1   +21.712, E3 +594650.346}
SPL {X  -162.820, Y  +439.933, Z    +0.000, E1   +21.690, E3 +594663.627}
SPL {X  -162.820, Y  +437.628, Z    +0.000, E1   +21.678, E3 +594675.815}
SPL {X  -162.820, Y  +434.473, Z    +0.000, E1   +21.747, E3 +594691.911}
SPL {X  -162.820, Y  +431.492, Z    +0.000, E1   +21.686, E3 +594707.860}
SPL {X  -162.820, Y  +429.074, Z    +0.000, E1   +21.710, E3 +594720.312}
SPL {X  -162.820, Y  +426.023, Z    +0.000, E1   +21.718, E3 +594736.380}
SPL {X  -162.820, Y  +422.986, Z    +0.000, E1   +21.685, E3 +594752.427}
SPL {X  -162.820, Y  +420.528, Z    +0.000, E1   +21.706, E3 +594765.077}
SPL {X  -162.820, Y  +418.116, Z    +0.000, E1   +21.761, E3 +594777.224}
SPL {X  -162.820, Y  +416.127, Z    +0.000, E1   +21.715, E3 +594787.929}
SPL {X  -162.820, Y  +414.361, Z    +0.000, E1   +21.613, E3 +594798.117}
SPL {X  -162.820, Y  +412.134, Z    +0.000, E1   +21.697, E3 +594809.061}
SPL {X  -162.820, Y  +409.248, Z    +0.000, E1   +21.741, E3 +594823.997}
SPL {X  -162.820, Y  +406.238, Z    +0.000, E1   +21.697, E3 +594839.965}
SPL {X  -162.820, Y  +404.001, Z    +0.000, E1   +21.723, E3 +594851.394}
SPL {X  -162.820, Y  +402.223, Z    +0.000, E1   +21.697, E3 +594860.879}
SPL {X  -162.820, Y  +400.348, Z    +0.000, E1   +21.713, E3 +594870.605}
SPL {X  -162.820, Y  +398.298, Z    +0.000, E1   +21.721, E3 +594881.221}
SPL {X  -162.820, Y  +396.371, Z    +0.000, E1   +21.713, E3 +594891.403}
SPL {X  -162.820, Y  +394.508, Z    +0.000, E1   +21.616, E3 +594901.958}
SPL {X  -162.820, Y  +392.435, Z    +0.000, E1   +21.681, E3 +594912.312}
SPL {X  -162.820, Y  +389.390, Z    +0.000, E1   +21.742, E3 +594927.918}
SPL {X  -162.820, Y  +386.818, Z    +0.000, E1   +21.679, E3 +594941.677}
SPL {X  -162.820, Y  +384.697, Z    +0.000, E1   +21.693, E3 +594952.747}
SPL {X  -162.820, Y  +382.288, Z    +0.000, E1   +21.742, E3 +594964.871}
SPL {X  -162.820, Y  +380.381, Z    +0.000, E1   +21.655, E3 +594975.596}
SPL {X  -162.808, Y  +378.512, Z    +0.000, E1   +21.736, E3 +594984.648}
SPL {X  -162.776, Y  +376.710, Z    +0.000, E1   +21.698, E3 +594994.448}
SPL {X  -162.707, Y  +374.438, Z    +0.000, E1   +21.688, E3 +595006.451}
SPL {X  -162.607, Y  +372.171, Z    +0.000, E1   +21.692, E3 +595018.251}
SPL {X  -162.494, Y  +370.197, Z    +0.000, E1   +21.655, E3 +595028.877}
SPL {X  -162.349, Y  +368.131, Z    +0.000, E1   +21.624, E3 +595039.995}
SPL {X  -162.161, Y  +365.866, Z    +0.000, E1   +21.642, E3 +595051.680}
SPL {X  -161.651, Y  +361.024, Z    +0.000, E1   +22.970, E3 +595065.104}
SPL {X  -160.281, Y  +351.857, Z    +0.000, E1   +24.243, E3 +595100.443}
ENDSPLINE

SPLINE
SPL {X  -161.833, Y  +362.603, Z    +0.000, E1   +17.021, E3 +595115.139}
ENDSPLINE

SPLINE
SPL {X  -160.786, Y  +354.842, Z    +0.000, E1   +19.274, E3 +595147.294}
ENDSPLINE

SPLINE
SPL {X  -162.485, Y  +370.062, Z    +0.000, E1   +10.606, E3 +595153.672}
SPL {X  -162.820, Y  +381.311, Z    +0.000, E1    +4.054, E3 +595144.028}
SPL {X  -162.820, Y  +390.142, Z    +0.000, E1    -2.185, E3 +595144.356}
SPL {X  -162.820, Y  +393.415, Z    +0.000, E1    -4.587, E3 +595149.463}
SPL {X  -162.820, Y  +399.630, Z    +0.000, E1    -9.426, E3 +595151.393}
SPL {X  -162.820, Y  +408.127, Z    +0.000, E1   -18.417, E3 +595137.681}
SPL {X  -162.820, Y  +420.083, Z    +0.000, E1   -24.325, E3 +595158.157}
SPL {X  -162.820, Y  +428.527, Z    +0.000, E1   -26.988, E3 +595175.449}
SPL {X  -162.820, Y  +431.336, Z    +0.000, E1   -24.162, E3 +595205.659}
SPL {X  -162.820, Y  +432.048, Z    +0.000, E1   -22.832, E3 +595220.162}
SPL {X  -162.820, Y  +434.888, Z    +0.000, E1   -22.823, E3 +595234.112}
SPL {X  -162.820, Y  +436.834, Z    +0.000, E1   -22.779, E3 +595244.072}
SPL {X  -162.820, Y  +438.868, Z    +0.000, E1   -22.837, E3 +595253.726}
SPL {X  -162.820, Y  +441.351, Z    +0.000, E1   -22.805, E3 +595266.301}
SPL {X  -162.820, Y  +443.809, Z    +0.000, E1   -22.804, E3 +595278.467}
SPL {X  -162.820, Y  +446.105, Z    +0.000, E1   -22.815, E3 +595289.709}
SPL {X  -162.820, Y  +447.974, Z    +0.000, E1   -22.856, E3 +595298.612}
SPL {X  -162.820, Y  +449.911, Z    +0.000, E1   -22.774, E3 +595308.887}
SPL {X  -162.820, Y  +451.861, Z    +0.000, E1   -22.750, E3 +595318.734}
SPL {X  -162.820, Y  +454.167, Z    +0.000, E1   -22.842, E3 +595329.464}
SPL {X  -162.820, Y  +456.529, Z    +0.000, E1   -22.855, E3 +595340.992}
SPL {X  -162.820, Y  +458.725, Z    +0.000, E1   -22.793, E3 +595352.397}
SPL {X  -162.820, Y  +461.700, Z    +0.000, E1   -22.822, E3 +595367.019}
SPL {X  -162.820, Y  +464.633, Z    +0.000, E1   -22.813, E3 +595381.516}
SPL {X  -162.820, Y  +467.913, Z    +0.000, E1   -22.879, E3 +595397.355}
SPL {X  -162.820, Y  +470.892, Z    +0.000, E1   -22.837, E3 +595412.245}
SPL {X  -162.820, Y  +472.726, Z    +0.000, E1   -22.777, E3 +595421.783}
SPL {X  -162.820, Y  +475.118, Z    +0.000, E1   -22.777, E3 +595433.755}
SPL {X  -162.820, Y  +478.177, Z    +0.000, E1   -22.834, E3 +595448.447}
SPL {X  -162.820, Y  +481.034, Z    +0.000, E1   -22.831, E3 +595462.585}
SPL {X  -162.820, Y  +483.391, Z    +0.000, E1   -22.793, E3 +595474.521}
SPL {X  -162.820, Y  +486.307, Z    +0.000, E1   -22.833, E3 +595488.775}
SPL {X  -162.820, Y  +489.750, Z    +0.000, E1   -22.832, E3 +595505.845}
SPL {X  -162.820, Y  +493.233, Z    +0.000, E1   -22.844, E3 +595522.982}
SPL {X  -162.820, Y  +496.150, Z    +0.000, E1   -22.796, E3 +595537.701}
SPL {X  -162.820, Y  +498.661, Z    +0.000, E1   -22.828, E3 +595549.882}
SPL {X  -162.820, Y  +501.761, Z    +0.000, E1   -22.820, E3 +595565.451}
SPL {X  -162.820, Y  +505.323, Z    +0.000, E1   -22.838, E3 +595582.898}
SPL {X  -162.820, Y  +508.611, Z    +0.000, E1   -22.838, E3 +595599.160}
SPL {X  -162.820, Y  +511.620, Z    +0.000, E1   -22.791, E3 +595614.404}
SPL {X  -162.820, Y  +513.873, Z    +0.000, E1   -22.800, E3 +595625.376}
SPL {X  -162.820, Y  +516.100, Z    +0.000, E1   -22.809, E3 +595636.453}
SPL {X  -162.820, Y  +518.662, Z    +0.000, E1   -22.847, E3 +595648.751}
SPL {X  -162.820, Y  +520.641, Z    +0.000, E1   -22.790, E3 +595658.992}
SPL {X  -162.820, Y  +523.535, Z    +0.000, E1   -22.857, E3 +595672.961}
SPL {X  -162.820, Y  +526.661, Z    +0.000, E1   -22.801, E3 +595688.785}
SPL {X  -162.820, Y  +528.725, Z    +0.000, E1   -22.770, E3 +595699.154}
SPL {X  -162.820, Y  +530.303, Z    +0.000, E1   -22.798, E3 +595706.774}
SPL {X  -162.820, Y  +532.614, Z    +0.000, E1   -22.828, E3 +595718.042}
SPL {X  -162.820, Y  +534.838, Z    +0.000, E1   -22.864, E3 +595728.671}
SPL {X  -162.820, Y  +536.882, Z    +0.000, E1   -22.782, E3 +595739.526}
SPL {X  -162.820, Y  +539.194, Z    +0.000, E1   -22.826, E3 +595750.574}
SPL {X  -162.820, Y  +541.555, Z    +0.000, E1   -22.817, E3 +595762.389}
SPL {X  -162.820, Y  +543.728, Z    +0.000, E1   -22.799, E3 +595773.246}
SPL {X  -162.820, Y  +545.925, Z    +0.000, E1   -22.803, E3 +595784.116}
SPL {X  -162.820, Y  +548.328, Z    +0.000, E1   -22.796, E3 +595796.112}
SPL {X  -162.820, Y  +551.027, Z    +0.000, E1   -22.819, E3 +595809.305}
SPL {X  -162.820, Y  +553.721, Z    +0.000, E1   -22.807, E3 +595822.749}
SPL {X  -162.820, Y  +556.430, Z    +0.000, E1   -22.821, E3 +595836.045}
SPL {X  -162.820, Y  +558.974, Z    +0.000, E1   -22.806, E3 +595848.745}
SPL {X  -162.820, Y  +562.171, Z    +0.000, E1   -22.845, E3 +595864.443}
SPL {X  -162.820, Y  +565.170, Z    +0.000, E1   -22.801, E3 +595879.456}
SPL {X  -162.820, Y  +567.308, Z    +0.000, E1   -22.750, E3 +595890.472}
SPL {X  -162.820, Y  +570.378, Z    +0.000, E1   -22.843, E3 +595905.096}
SPL {X  -162.820, Y  +573.634, Z    +0.000, E1   -22.827, E3 +595921.240}
SPL {X  -162.820, Y  +576.228, Z    +0.000, E1   -22.814, E3 +595934.136}
SPL {X  -162.820, Y  +578.553, Z    +0.000, E1   -22.801, E3 +595945.752}
SPL {X  -162.820, Y  +581.064, Z    +0.000, E1   -22.823, E3 +595958.036}
SPL {X  -162.820, Y  +583.435, Z    +0.000, E1   -22.808, E3 +595969.858}
SPL {X  -162.820, Y  +585.410, Z    +0.000, E1   -22.764, E3 +595979.994}
SPL {X  -162.820, Y  +587.676, Z    +0.000, E1   -22.853, E3 +595990.509}
SPL {X  -162.820, Y  +589.682, Z    +0.000, E1   -22.776, E3 +596001.038}
SPL {X  -162.820, Y  +591.720, Z    +0.000, E1   -22.868, E3 +596010.349}
SPL {X  -162.820, Y  +593.650, Z    +0.000, E1   -22.810, E3 +596020.419}
SPL {X  -162.820, Y  +595.830, Z    +0.000, E1   -22.828, E3 +596031.035}
SPL {X  -162.820, Y  +598.094, Z    +0.000, E1   -22.843, E3 +596042.148}
SPL {X  -162.820, Y  +600.420, Z    +0.000, E1   -22.826, E3 +596053.779}
SPL {X  -162.820, Y  +602.573, Z    +0.000, E1   -22.830, E3 +596064.364}
SPL {X  -162.820, Y  +604.828, Z    +0.000, E1   -22.784, E3 +596076.003}
SPL {X  -162.820, Y  +608.133, Z    +0.000, E1   -22.831, E3 +596092.121}
SPL {X  -162.820, Y  +611.103, Z    +0.000, E1   -22.785, E3 +596107.046}
SPL {X  -162.820, Y  +613.294, Z    +0.000, E1   -22.780, E3 +596117.919}
SPL {X  -162.820, Y  +615.356, Z    +0.000, E1   -22.799, E3 +596127.977}
SPL {X  -162.820, Y  +617.439, Z    +0.000, E1   -22.808, E3 +596138.235}
SPL {X  -162.820, Y  +619.665, Z    +0.000, E1   -22.817, E3 +596149.203}
SPL {X  -162.820, Y  +621.733, Z    +0.000, E1   -22.759, E3 +596159.927}
SPL {X  -162.820, Y  +624.076, Z    +0.000, E1   -22.774, E3 +596171.432}
SPL {X  -162.820, Y  +626.527, Z    +0.000, E1   -22.768, E3 +596183.675}
SPL {X  -162.820, Y  +629.758, Z    +0.000, E1   -22.800, E3 +596199.603}
SPL {X  -162.820, Y  +632.572, Z    +0.000, E1   -22.785, E3 +596213.453}
SPL {X  -162.820, Y  +634.507, Z    +0.000, E1   -22.784, E3 +596223.092}
SPL {X  -162.820, Y  +636.863, Z    +0.000, E1   -22.760, E3 +596235.014}
SPL {X  -162.820, Y  +639.254, Z    +0.000, E1   -22.767, E3 +596246.797}
SPL {X  -162.820, Y  +641.888, Z    +0.000, E1   -22.790, E3 +596259.744}
SPL {X  -162.820, Y  +644.915, Z    +0.000, E1   -22.818, E3 +596274.519}
SPL {X  -162.820, Y  +647.561, Z    +0.000, E1   -22.705, E3 +596288.561}
SPL {X  -162.820, Y  +649.758, Z    +0.000, E1   -22.780, E3 +596298.751}
SPL {X  -162.820, Y  +651.708, Z    +0.000, E1   -22.810, E3 +596308.246}
SPL {X  -162.820, Y  +653.898, Z    +0.000, E1   -22.796, E3 +596319.166}
SPL {X  -162.820, Y  +656.161, Z    +0.000, E1   -22.812, E3 +596330.288}
SPL {X  -162.820, Y  +658.384, Z    +0.000, E1   -22.822, E3 +596341.154}
SPL {X  -162.820, Y  +660.215, Z    +0.000, E1   -22.649, E3 +596351.745}
SPL {X  -162.820, Y  +662.823, Z    +0.000, E1   -22.799, E3 +596363.453}
SPL {X  -162.820, Y  +665.112, Z    +0.000, E1   -22.835, E3 +596374.507}
SPL {X  -162.820, Y  +667.016, Z    +0.000, E1   -22.823, E3 +596383.936}
SPL {X  -162.820, Y  +668.960, Z    +0.000, E1   -22.773, E3 +596394.103}
SPL {X  -162.820, Y  +672.333, Z    +0.000, E1   -22.837, E3 +596410.439}
SPL {X  -162.812, Y  +675.071, Z    +0.000, E1   -22.742, E3 +596424.584}
SPL {X  -162.773, Y  +677.428, Z    +0.000, E1   -22.762, E3 +596436.182}
SPL {X  -162.691, Y  +679.987, Z    +0.000, E1   -22.794, E3 +596448.595}
SPL {X  -162.559, Y  +682.717, Z    +0.000, E1   -22.726, E3 +596462.778}
SPL {X  -162.349, Y  +685.880, Z    +0.000, E1   -22.738, E3 +596478.380}
SPL {X  -162.164, Y  +688.106, Z    +0.000, E1   -22.661, E3 +596489.900}
SPL {X  -161.938, Y  +690.422, Z    +0.000, E1   -22.769, E3 +596500.575}
SPL {X  -161.065, Y  +697.344, Z    +0.000, E1   -25.698, E3 +596509.695}
SPL {X  -158.553, Y  +710.529, Z    +0.000, E1   -30.890, E3 +596523.591}
ENDSPLINE

SPLINE
SPL {X  -161.215, Y  +696.305, Z    +0.000, E1   -20.575, E3 +596550.172}
SPL {X  -161.691, Y  +692.643, Z    +0.000, E1   -17.369, E3 +596566.360}
SPL {X  -162.534, Y  +683.153, Z    +0.000, E1   -10.475, E3 +596591.827}
SPL {X  -162.820, Y  +670.105, Z    +0.000, E1    -2.484, E3 +596584.474}
SPL {X  -162.820, Y  +665.819, Z    +0.000, E1    +0.492, E3 +596586.770}
SPL {X  -162.820, Y  +661.883, Z    +0.000, E1    +3.373, E3 +596591.247}
SPL {X  -162.820, Y  +655.163, Z    +0.000, E1    +8.702, E3 +596590.846}
SPL {X  -162.820, Y  +634.515, Z    +0.000, E1   +26.439, E3 +596583.259}
ENDSPLINE

SPLINE
SPL {X  -162.820, Y  +638.080, Z    +0.000, E1   +18.858, E3 +596613.223}
ENDSPLINE

SPLINE
SPL {X  -162.820, Y  +623.278, Z    +0.000, E1   +28.723, E3 +596614.794}
SPL {X  -162.820, Y  +618.658, Z    +0.000, E1   +26.841, E3 +596643.403}
ENDSPLINE

SPLINE
SPL {X  -162.820, Y  +623.685, Z    +0.000, E1   +22.346, E3 +596655.710}
ENDSPLINE

SPLINE
SPL {X  -162.820, Y  +621.304, Z    +0.000, E1   +22.259, E3 +596668.525}
SPL {X  -162.820, Y  +618.758, Z    +0.000, E1   +22.239, E3 +596681.676}
SPL {X  -162.820, Y  +616.062, Z    +0.000, E1   +22.275, E3 +596695.096}
SPL {X  -162.820, Y  +613.536, Z    +0.000, E1   +22.242, E3 +596708.218}
SPL {X  -162.820, Y  +610.461, Z    +0.000, E1   +22.264, E3 +596723.849}
SPL {X  -162.820, Y  +607.796, Z    +0.000, E1   +22.261, E3 +596737.220}
SPL {X  -162.820, Y  +605.178, Z    +0.000, E1   +22.267, E3 +596750.704}
SPL {X  -162.820, Y  +602.350, Z    +0.000, E1   +22.224, E3 +596765.321}
SPL {X  -162.820, Y  +599.842, Z    +0.000, E1   +22.298, E3 +596777.473}
SPL {X  -162.820, Y  +597.194, Z    +0.000, E1   +22.253, E3 +596791.394}
SPL {X  -162.820, Y  +594.115, Z    +0.000, E1   +22.273, E3 +596806.922}
SPL {X  -162.820, Y  +591.721, Z    +0.000, E1   +22.239, E3 +596819.237}
SPL {X  -162.820, Y  +589.492, Z    +0.000, E1   +22.304, E3 +596830.098}
SPL {X  -162.820, Y  +587.447, Z    +0.000, E1   +22.279, E3 +596840.627}
SPL {X  -162.820, Y  +585.192, Z    +0.000, E1   +22.298, E3 +596852.038}
SPL {X  -162.820, Y  +582.610, Z    +0.000, E1   +22.234, E3 +596865.661}
SPL {X  -162.820, Y  +580.317, Z    +0.000, E1   +22.300, E3 +596876.715}
SPL {X  -162.820, Y  +578.878, Z    +0.000, E1   +22.272, E3 +596884.224}
SPL {X  -162.820, Y  +576.856, Z    +0.000, E1   +22.233, E3 +596894.983}
SPL {X  -162.820, Y  +573.830, Z    +0.000, E1   +22.272, E3 +596910.119}
SPL {X  -162.820, Y  +570.852, Z    +0.000, E1   +22.234, E3 +596925.578}
SPL {X  -162.820, Y  +568.608, Z    +0.000, E1   +22.253, E3 +596936.711}
SPL {X  -162.820, Y  +565.838, Z    +0.000, E1   +22.271, E3 +596950.943}
SPL {X  -162.820, Y  +562.162, Z    +0.000, E1   +22.252, E3 +596969.760}
SPL {X  -162.820, Y  +558.919, Z    +0.000, E1   +22.286, E3 +596985.923}
SPL {X  -162.820, Y  +555.548, Z    +0.000, E1   +22.322, E3 +597002.832}
SPL {X  -162.820, Y  +552.787, Z    +0.000, E1   +22.213, E3 +597017.630}
SPL {X  -162.820, Y  +550.871, Z    +0.000, E1   +22.229, E3 +597027.224}
SPL {X  -162.820, Y  +548.168, Z    +0.000, E1   +22.298, E3 +597040.560}
SPL {X  -162.820, Y  +545.860, Z    +0.000, E1   +22.216, E3 +597052.818}
SPL {X  -162.820, Y  +543.558, Z    +0.000, E1   +22.285, E3 +597064.048}
SPL {X  -162.820, Y  +540.968, Z    +0.000, E1   +22.274, E3 +597077.321}
SPL {X  -162.820, Y  +538.512, Z    +0.000, E1   +22.287, E3 +597089.633}
SPL {X  -162.820, Y  +535.523, Z    +0.000, E1   +22.266, E3 +597105.249}
SPL {X  -162.820, Y  +531.757, Z    +0.000, E1   +22.276, E3 +597124.303}
SPL {X  -162.820, Y  +527.980, Z    +0.000, E1   +22.326, E3 +597143.134}
SPL {X  -162.820, Y  +524.599, Z    +0.000, E1   +22.287, E3 +597160.532}
SPL {X  -162.820, Y  +522.011, Z    +0.000, E1   +22.282, E3 +597173.609}
SPL {X  -162.820, Y  +519.457, Z    +0.000, E1   +22.481, E3 +597184.898}
SPL {X  -162.820, Y  +505.859, Z    +0.000, E1   +28.367, E3 +597199.381}
SPL {X  -162.820, Y  +504.131, Z    +0.000, E1   +27.325, E3 +597213.519}
SPL {X  -162.820, Y  +503.215, Z    +0.000, E1   +26.369, E3 +597224.205}
SPL {X  -162.820, Y  +502.265, Z    +0.000, E1   +25.287, E3 +597236.688}
SPL {X  -162.820, Y  +501.060, Z    +0.000, E1   +24.081, E3 +597251.428}
SPL {X  -162.820, Y  +500.336, Z    +0.000, E1   +23.110, E3 +597262.568}
SPL {X  -162.820, Y  +499.240, Z    +0.000, E1   +22.316, E3 +597274.879}
SPL {X  -162.820, Y  +498.027, Z    +0.000, E1   +21.516, E3 +597287.786}
SPL {X  -162.820, Y  +495.897, Z    +0.000, E1   +21.662, E3 +597297.706}
SPL {X  -162.820, Y  +493.717, Z    +0.000, E1   +21.704, E3 +597308.813}
SPL {X  -162.820, Y  +491.396, Z    +0.000, E1   +21.707, E3 +597320.937}
SPL {X  -162.820, Y  +488.560, Z    +0.000, E1   +21.695, E3 +597336.046}
SPL {X  -162.820, Y  +485.661, Z    +0.000, E1   +21.712, E3 +597350.931}
SPL {X  -162.820, Y  +483.668, Z    +0.000, E1   +21.664, E3 +597361.759}
SPL {X  -162.820, Y  +481.739, Z    +0.000, E1   +21.704, E3 +597371.473}
SPL {X  -162.820, Y  +479.894, Z    +0.000, E1   +21.695, E3 +597381.260}
SPL {X  -162.820, Y  +477.685, Z    +0.000, E1   +21.656, E3 +597393.198}
SPL {X  -162.820, Y  +475.419, Z    +0.000, E1   +21.711, E3 +597404.550}
SPL {X  -162.820, Y  +473.301, Z    +0.000, E1   +21.712, E3 +597415.647}
SPL {X  -162.820, Y  +470.965, Z    +0.000, E1   +21.700, E3 +597427.992}
SPL {X  -162.820, Y  +469.036, Z    +0.000, E1   +21.695, E3 +597438.036}
SPL {X  -162.820, Y  +467.138, Z    +0.000, E1   +21.678, E3 +597448.208}
SPL {X  -162.820, Y  +465.011, Z    +0.000, E1   +21.692, E3 +597459.190}
SPL {X  -162.820, Y  +462.669, Z    +0.000, E1   +21.752, E3 +597470.971}
SPL {X  -162.820, Y  +460.725, Z    +0.000, E1   +21.689, E3 +597481.584}
SPL {X  -162.820, Y  +458.666, Z    +0.000, E1   +21.695, E3 +597492.396}
SPL {X  -162.820, Y  +456.431, Z    +0.000, E1   +21.708, E3 +597503.924}
SPL {X  -162.820, Y  +454.628, Z    +0.000, E1   +21.674, E3 +597513.642}
SPL {X  -162.820, Y  +452.690, Z    +0.000, E1   +21.773, E3 +597522.917}
SPL {X  -162.820, Y  +450.610, Z    +0.000, E1   +21.698, E3 +597534.515}
SPL {X  -162.820, Y  +448.170, Z    +0.000, E1   +21.667, E3 +597547.536}
SPL {X  -162.820, Y  +446.246, Z    +0.000, E1   +21.696, E3 +597557.354}
SPL {X  -162.820, Y  +443.784, Z    +0.000, E1   +21.713, E3 +597570.140}
SPL {X  -162.820, Y  +440.567, Z    +0.000, E1   +21.731, E3 +597586.980}
SPL {X  -162.820, Y  +437.628, Z    +0.000, E1   +21.678, E3 +597602.644}
SPL {X  -162.820, Y  +435.262, Z    +0.000, E1   +21.727, E3 +597614.580}
SPL {X  -162.820, Y  +433.510, Z    +0.000, E1   +21.692, E3 +597623.994}
SPL {X  -162.820, Y  +431.492, Z    +0.000, E1   +21.686, E3 +597634.689}
SPL {X  -162.820, Y  +429.074, Z    +0.000, E1   +21.710, E3 +597647.141}
SPL {X  -162.820, Y  +427.020, Z    +0.000, E1   +21.674, E3 +597658.142}
SPL {X  -162.820, Y  +424.525, Z    +0.000, E1   +21.712, E3 +597671.055}
SPL {X  -162.820, Y  +421.144, Z    +0.000, E1   +21.719, E3 +597688.722}
SPL {X  -162.820, Y  +418.116, Z    +0.000, E1   +21.761, E3 +597704.053}
SPL {X  -162.820, Y  +416.127, Z    +0.000, E1   +21.715, E3 +597714.759}
SPL {X  -162.820, Y  +414.361, Z    +0.000, E1   +21.613, E3 +597724.946}
SPL {X  -162.820, Y  +411.450, Z    +0.000, E1   +21.710, E3 +597739.519}
SPL {X  -162.820, Y  +408.590, Z    +0.000, E1   +21.735, E3 +597754.145}
SPL {X  -162.820, Y  +406.238, Z    +0.000, E1   +21.697, E3 +597766.794}
SPL {X  -162.820, Y  +403.166, Z    +0.000, E1   +21.746, E3 +597782.600}
SPL {X  -162.820, Y  +400.348, Z    +0.000, E1   +21.713, E3 +597797.435}
SPL {X  -162.820, Y  +398.298, Z    +0.000, E1   +21.721, E3 +597808.050}
SPL {X  -162.820, Y  +396.371, Z    +0.000, E1   +21.713, E3 +597818.232}
SPL {X  -162.820, Y  +394.508, Z    +0.000, E1   +21.616, E3 +597828.787}
SPL {X  -162.820, Y  +392.435, Z    +0.000, E1   +21.681, E3 +597839.141}
SPL {X  -162.820, Y  +389.390, Z    +0.000, E1   +21.742, E3 +597854.748}
SPL {X  -162.820, Y  +386.818, Z    +0.000, E1   +21.679, E3 +597868.506}
SPL {X  -162.820, Y  +384.697, Z    +0.000, E1   +21.693, E3 +597879.577}
SPL {X  -162.820, Y  +382.288, Z    +0.000, E1   +21.742, E3 +597891.700}
SPL {X  -162.817, Y  +379.520, Z    +0.000, E1   +21.723, E3 +597906.538}
SPL {X  -162.776, Y  +376.710, Z    +0.000, E1   +21.698, E3 +597921.277}
SPL {X  -162.707, Y  +374.438, Z    +0.000, E1   +21.688, E3 +597933.281}
SPL {X  -162.607, Y  +372.171, Z    +0.000, E1   +21.692, E3 +597945.080}
SPL {X  -162.494, Y  +370.197, Z    +0.000, E1   +21.655, E3 +597955.707}
SPL {X  -162.349, Y  +368.131, Z    +0.000, E1   +21.624, E3 +597966.825}
SPL {X  -162.161, Y  +365.866, Z    +0.000, E1   +21.642, E3 +597978.510}
SPL {X  -161.651, Y  +361.024, Z    +0.000, E1   +22.970, E3 +597991.933}
SPL {X  -160.281, Y  +351.857, Z    +0.000, E1   +24.243, E3 +598027.272}
ENDSPLINE

SPLINE
SPL {X  -161.833, Y  +362.603, Z    +0.000, E1   +17.021, E3 +598041.968}
ENDSPLINE

SPLINE
SPL {X  -160.786, Y  +354.842, Z    +0.000, E1   +19.274, E3 +598074.124}
ENDSPLINE

